C03633=1071.064,-119.142,443.657,172.455,21.905,153.991
C03634=1071.070,-118.892,443.648,172.457,21.906,153.991
C03635=1071.076,-118.643,443.638,172.457,21.907,153.991
C03636=1071.082,-118.393,443.629,172.459,21.908,153.991
C03637=1071.088,-118.143,443.619,172.461,21.909,153.991
C03638=1071.094,-117.893,443.610,172.463,21.910,153.991
C03639=1071.100,-117.643,443.601,172.464,21.911,153.990
C03640=1071.106,-117.393,443.591,172.466,21.912,153.990
C03641=1071.112,-117.143,443.582,172.468,21.913,153.990
C03642=1071.119,-116.893,443.572,172.469,21.914,153.990
C03643=1071.125,-116.644,443.563,172.471,21.915,153.990
C03644=1071.130,-116.395,443.553,172.473,21.916,153.990
C03645=1071.137,-116.145,443.544,172.475,21.917,153.990
C03646=1071.143,-115.895,443.535,172.476,21.918,153.990
C03647=1071.150,-115.646,443.525,172.478,21.919,153.990
C03648=1071.156,-115.396,443.516,172.479,21.920,153.990
C03649=1071.162,-115.146,443.506,172.480,21.921,153.990
C03650=1071.168,-114.896,443.497,172.482,21.922,153.990
C03651=1071.174,-114.646,443.487,172.484,21.923,153.990
C03652=1071.181,-114.367,443.476,172.486,21.924,153.990
C03653=1071.188,-114.087,443.466,172.488,21.925,153.989
C03654=1071.195,-113.808,443.455,172.490,21.927,153.989
C03655=1071.201,-113.528,443.443,172.492,21.927,153.989
C03656=1071.208,-113.278,443.434,172.493,21.929,153.989
C03657=1071.214,-113.029,443.424,172.495,21.930,153.989
C03658=1071.220,-112.779,443.415,172.497,21.931,153.989
C03659=1071.226,-112.529,443.405,172.498,21.932,153.989
C03660=1071.232,-112.280,443.396,172.500,21.933,153.989
C03661=1071.238,-112.030,443.386,172.502,21.934,153.989
C03662=1071.244,-111.780,443.377,172.502,21.935,153.989
C03663=1071.250,-111.531,443.367,172.504,21.936,153.989
C03664=1071.257,-111.281,443.357,172.506,21.937,153.989
C03665=1071.263,-111.032,443.347,172.508,21.938,153.989
C03666=1071.269,-110.782,443.338,172.509,21.939,153.989
C03667=1071.274,-110.532,443.328,172.511,21.940,153.989
C03668=1071.281,-110.282,443.318,172.512,21.942,153.989
C03669=1071.287,-110.032,443.309,172.514,21.942,153.989
C03670=1071.293,-109.782,443.299,172.516,21.944,153.989
C03671=1071.299,-109.533,443.289,172.517,21.945,153.989
C03672=1071.306,-109.283,443.279,172.519,21.946,153.989
C03673=1071.312,-109.034,443.270,172.521,21.947,153.989
C03674=1071.318,-108.784,443.260,172.523,21.948,153.989
C03675=1071.324,-108.534,443.250,172.524,21.950,153.989
C03676=1071.330,-108.284,443.241,172.526,21.950,153.988
C03677=1071.336,-108.035,443.230,172.527,21.952,153.988
C03678=1071.342,-107.785,443.220,172.529,21.953,153.988
C03679=1071.348,-107.535,443.211,172.531,21.954,153.988
C03680=1071.354,-107.285,443.201,172.532,21.955,153.988
C03681=1071.361,-107.035,443.192,172.533,21.956,153.988
C03682=1071.367,-106.786,443.181,172.535,21.957,153.988
C03683=1071.373,-106.536,443.171,172.536,21.959,153.988
C03684=1071.379,-106.286,443.162,172.538,21.960,153.988
C03685=1071.385,-106.037,443.152,172.540,21.961,153.988
C03686=1071.391,-105.787,443.142,172.541,21.962,153.988
C03687=1071.397,-105.537,443.132,172.543,21.964,153.988
C03688=1071.403,-105.287,443.122,172.545,21.964,153.988
C03689=1071.409,-105.038,443.113,172.546,21.966,153.988
C03690=1071.416,-104.788,443.102,172.548,21.967,153.988
C03691=1071.422,-104.538,443.092,172.550,21.968,153.988
C03692=1071.428,-104.288,443.082,172.551,21.969,153.988
C03693=1071.434,-104.039,443.072,172.553,21.971,153.988
C03694=1071.441,-103.789,443.062,172.554,21.972,153.988
C03695=1071.446,-103.539,443.052,172.556,21.973,153.988
C03696=1071.452,-103.290,443.042,172.558,21.974,153.988
C03697=1071.459,-103.040,443.032,172.559,21.976,153.988
C03698=1071.464,-102.790,443.022,172.561,21.977,153.988
C03699=1071.470,-102.541,443.012,172.563,21.978,153.988
C03700=1071.477,-102.291,443.002,172.564,21.979,153.988
C03701=1071.483,-102.041,442.993,172.566,21.981,153.988
C03702=1071.489,-101.791,442.982,172.568,21.982,153.988
C03703=1071.495,-101.542,442.972,172.569,21.983,153.988
C03704=1071.501,-101.292,442.963,172.571,21.985,153.988
C03705=1071.507,-101.042,442.952,172.573,21.986,153.988
C03706=1071.513,-100.792,442.942,172.574,21.987,153.988
C03707=1071.520,-100.543,442.932,172.576,21.988,153.988
C03708=1071.525,-100.293,442.921,172.577,21.990,153.988
C03709=1071.532,-100.043,442.912,172.579,21.991,153.988
C03710=1071.538,-99.794,442.902,172.580,21.992,153.988
C03711=1071.543,-99.543,442.891,172.581,21.993,153.988
C03712=1071.550,-99.294,442.881,172.583,21.994,153.988
C03713=1071.556,-99.045,442.872,172.584,21.996,153.988
C03714=1071.562,-98.795,442.861,172.586,21.997,153.988
C03715=1071.569,-98.545,442.851,172.588,21.998,153.988
C03716=1071.575,-98.263,442.839,172.590,22.000,153.988
C03717=1071.583,-97.981,442.828,172.592,22.001,153.988
C03718=1071.589,-97.699,442.817,172.593,22.003,153.988
C03719=1071.596,-97.417,442.805,172.595,22.004,153.988
C03720=1071.602,-97.167,442.795,172.596,22.006,153.988
C03721=1071.608,-96.918,442.784,172.598,22.007,153.988
C03722=1071.614,-96.668,442.775,172.600,22.008,153.988
C03723=1071.620,-96.418,442.764,172.601,22.010,153.988
C03724=1071.626,-96.169,442.754,172.603,22.011,153.988
C03725=1071.632,-95.919,442.743,172.604,22.012,153.988
C03726=1071.638,-95.670,442.732,172.606,22.014,153.988
C03727=1071.644,-95.420,442.723,172.608,22.015,153.988
C03728=1071.650,-95.170,442.712,172.609,22.017,153.988
C03729=1071.656,-94.920,442.702,172.611,22.018,153.988
C03730=1071.662,-94.670,442.691,172.612,22.019,153.988
C03731=1071.668,-94.421,442.682,172.614,22.021,153.988
C03732=1071.674,-94.171,442.671,172.615,22.022,153.988
C03733=1071.680,-93.921,442.661,172.617,22.023,153.988
C03734=1071.686,-93.672,442.650,172.619,22.025,153.988
C03735=1071.692,-93.423,442.640,172.620,22.027,153.988
C03736=1071.698,-93.172,442.629,172.622,22.028,153.988
C03737=1071.704,-92.922,442.619,172.623,22.030,153.988
C03738=1071.711,-92.673,442.608,172.625,22.031,153.988
C03739=1071.716,-92.423,442.598,172.626,22.032,153.988
C03740=1071.723,-92.174,442.588,172.628,22.034,153.988
C03741=1071.728,-91.924,442.578,172.630,22.035,153.988
C03742=1071.735,-91.674,442.567,172.631,22.036,153.989
C03743=1071.741,-91.424,442.556,172.633,22.038,153.989
C03744=1071.746,-91.174,442.546,172.634,22.039,153.989
C03745=1071.753,-90.925,442.536,172.636,22.041,153.989
C03746=1071.759,-90.676,442.525,172.637,22.042,153.989
C03747=1071.765,-90.426,442.515,172.639,22.044,153.989
C03748=1071.771,-90.176,442.504,172.640,22.045,153.989
C03749=1071.777,-89.926,442.493,172.642,22.047,153.989
C03750=1071.783,-89.676,442.484,172.644,22.048,153.989
C03751=1071.789,-89.427,442.473,172.645,22.049,153.989
C03752=1071.796,-89.177,442.462,172.647,22.051,153.989
C03753=1071.801,-88.927,442.451,172.648,22.053,153.989
C03754=1071.807,-88.677,442.441,172.650,22.054,153.989
C03755=1071.813,-88.428,442.431,172.651,22.055,153.989
C03756=1071.820,-88.178,442.420,172.653,22.057,153.989
C03757=1071.825,-87.928,442.409,172.654,22.059,153.989
C03758=1071.832,-87.679,442.399,172.656,22.060,153.989
C03759=1071.837,-87.429,442.388,172.658,22.061,153.989
C03760=1071.844,-87.179,442.378,172.659,22.063,153.989
C03761=1071.850,-86.930,442.367,172.661,22.064,153.989
C03762=1071.856,-86.680,442.357,172.662,22.066,153.989
C03763=1071.862,-86.431,442.346,172.664,22.068,153.989
C03764=1071.868,-86.180,442.335,172.665,22.069,153.989
C03765=1071.874,-85.931,442.324,172.667,22.070,153.989
C03766=1071.881,-85.682,442.314,172.668,22.072,153.989
C03767=1071.886,-85.432,442.303,172.670,22.074,153.990
C03768=1071.892,-85.181,442.292,172.671,22.075,153.990
C03769=1071.899,-84.932,442.282,172.673,22.076,153.990
C03770=1071.905,-84.683,442.271,172.675,22.078,153.990
C03771=1071.911,-84.433,442.260,172.676,22.080,153.990
C03772=1071.917,-84.183,442.250,172.678,22.081,153.990
C03773=1071.923,-83.934,442.239,172.679,22.082,153.990
C03774=1071.929,-83.683,442.228,172.681,22.084,153.990
C03775=1071.936,-83.434,442.218,172.682,22.086,153.990
C03776=1071.941,-83.184,442.207,172.684,22.087,153.990
C03777=1071.948,-82.934,442.196,172.685,22.088,153.990
C03778=1071.954,-82.685,442.186,172.687,22.090,153.990
C03779=1071.960,-82.436,442.175,172.689,22.092,153.990
C03780=1071.967,-82.156,442.163,172.691,22.093,153.990
C03781=1071.974,-81.877,442.150,172.692,22.095,153.990
C03782=1071.981,-81.597,442.138,172.694,22.097,153.990
C03783=1071.988,-81.317,442.127,172.696,22.099,153.990
C03784=1071.994,-81.067,442.116,172.698,22.100,153.990
C03785=1072.000,-80.818,442.105,172.699,22.102,153.990
C03786=1072.007,-80.568,442.094,172.701,22.104,153.991
C03787=1072.013,-80.318,442.083,172.702,22.105,153.991
C03788=1072.018,-80.069,442.073,172.704,22.107,153.991
C03789=1072.025,-79.819,442.061,172.705,22.108,153.991
C03790=1072.031,-79.569,442.051,172.707,22.110,153.991
C03791=1072.037,-79.320,442.040,172.708,22.112,153.991
C03792=1072.043,-79.070,442.029,172.710,22.113,153.991
C03793=1072.049,-78.820,442.018,172.711,22.115,153.991
C03794=1072.055,-78.571,442.007,172.713,22.116,153.991
C03795=1072.061,-78.321,441.996,172.714,22.118,153.991
C03796=1072.067,-78.071,441.985,172.716,22.120,153.991
C03797=1072.073,-77.821,441.974,172.717,22.121,153.991
C03798=1072.079,-77.571,441.963,172.719,22.123,153.992
C03799=1072.085,-77.322,441.952,172.720,22.124,153.992
C03800=1072.092,-77.072,441.941,172.722,22.126,153.992
C03801=1072.097,-76.822,441.930,172.723,22.128,153.992
C03802=1072.103,-76.573,441.920,172.725,22.130,153.992
C03803=1072.110,-76.323,441.908,172.726,22.131,153.992
C03804=1072.116,-76.074,441.897,172.728,22.133,153.992
C03805=1072.121,-75.824,441.886,172.729,22.134,153.992
C03806=1072.128,-75.574,441.875,172.731,22.136,153.992
C03807=1072.133,-75.325,441.864,172.732,22.138,153.992
C03808=1072.140,-75.075,441.853,172.734,22.140,153.992
C03809=1072.145,-74.825,441.842,172.735,22.141,153.992
C03810=1072.152,-74.575,441.830,172.737,22.143,153.993
C03811=1072.158,-74.325,441.820,172.738,22.144,153.993
C03812=1072.164,-74.076,441.809,172.741,22.147,153.993
C03813=1072.170,-73.826,441.797,172.742,22.148,153.993
C03814=1072.176,-73.577,441.786,172.743,22.150,153.993
C03815=1072.181,-73.327,441.775,172.745,22.152,153.993
C03816=1072.188,-73.077,441.764,172.746,22.154,153.993
C03817=1072.193,-72.828,441.753,172.748,22.155,153.993
C03818=1072.200,-72.577,441.742,172.749,22.157,153.993
C03819=1072.206,-72.329,441.730,172.751,22.159,153.993
C03820=1072.212,-72.079,441.719,172.752,22.160,153.993
C03821=1072.217,-71.829,441.707,172.754,22.162,153.994
C03822=1072.223,-71.579,441.696,172.755,22.164,153.994
C03823=1072.229,-71.330,441.685,172.757,22.165,153.994
C03824=1072.235,-71.080,441.674,172.758,22.167,153.994
C03825=1072.241,-70.831,441.663,172.759,22.169,153.994
C03826=1072.247,-70.580,441.651,172.761,22.171,153.994
C03827=1072.253,-70.331,441.639,172.762,22.173,153.994
C03828=1072.258,-70.082,441.628,172.764,22.175,153.994
C03829=1072.265,-69.832,441.617,172.765,22.176,153.995
C03830=1072.271,-69.582,441.606,172.767,22.178,153.995
C03831=1072.277,-69.332,441.594,172.768,22.180,153.995
C03832=1072.283,-69.083,441.583,172.770,22.182,153.995
C03833=1072.289,-68.832,441.572,172.772,22.184,153.995
C03834=1072.294,-68.583,441.561,172.774,22.185,153.995
C03835=1072.300,-68.334,441.549,172.775,22.187,153.995
C03836=1072.307,-68.084,441.538,172.776,22.189,153.995
C03837=1072.312,-67.834,441.527,172.778,22.191,153.995
C03838=1072.319,-67.585,441.515,172.779,22.193,153.995
C03839=1072.324,-67.335,441.504,172.781,22.194,153.996
C03840=1072.330,-67.085,441.492,172.782,22.196,153.996
C03841=1072.336,-66.836,441.481,172.784,22.198,153.996
C03842=1072.343,-66.586,441.469,172.785,22.200,153.996
C03843=1072.349,-66.337,441.458,172.786,22.202,153.996
C03844=1072.355,-66.059,441.445,172.788,22.204,153.996
C03845=1072.362,-65.782,441.432,172.790,22.206,153.996
C03846=1072.369,-65.504,441.419,172.792,22.208,153.996
C03847=1072.376,-65.227,441.407,172.793,22.210,153.997
C03848=1072.381,-64.977,441.395,172.794,22.212,153.997
C03849=1072.387,-64.727,441.384,172.796,22.214,153.997
C03850=1072.393,-64.478,441.373,172.797,22.215,153.997
C03851=1072.400,-64.228,441.361,172.799,22.217,153.997
C03852=1072.405,-63.978,441.349,172.801,22.219,153.997
C03853=1072.411,-63.728,441.338,172.802,22.221,153.997
C03854=1072.417,-63.479,441.326,172.804,22.223,153.997
C03855=1072.423,-63.229,441.315,172.805,22.225,153.998
C03856=1072.429,-62.980,441.304,172.807,22.227,153.998
C03857=1072.435,-62.730,441.292,172.808,22.229,153.998
C03858=1072.441,-62.481,441.280,172.810,22.230,153.998
C03859=1072.447,-62.231,441.269,172.811,22.232,153.998
C03860=1072.454,-61.981,441.257,172.812,22.234,153.998
C03861=1072.459,-61.731,441.245,172.814,22.236,153.998
C03862=1072.466,-61.482,441.233,172.815,22.238,153.999
C03863=1072.472,-61.232,441.223,172.817,22.240,153.999
C03864=1072.478,-60.983,441.211,172.818,22.242,153.999
C03865=1072.483,-60.733,441.199,172.820,22.243,153.999
C03866=1072.490,-60.483,441.187,172.821,22.245,153.999
C03867=1072.496,-60.233,441.176,172.823,22.247,153.999
C03868=1072.501,-59.984,441.164,172.825,22.249,153.999
C03869=1072.508,-59.734,441.152,172.826,22.251,153.999
C03870=1072.514,-59.485,441.141,172.828,22.253,154.000
C03871=1072.520,-59.235,441.129,172.829,22.255,154.000
C03872=1072.526,-58.985,441.117,172.830,22.257,154.000
C03873=1072.532,-58.736,441.106,172.832,22.258,154.000
C03874=1072.538,-58.486,441.094,172.833,22.260,154.000
C03875=1072.544,-58.236,441.082,172.835,22.262,154.000
C03876=1072.550,-57.987,441.070,172.836,22.264,154.000
C03877=1072.557,-57.737,441.059,172.838,22.266,154.001
C03878=1072.563,-57.488,441.047,172.839,22.268,154.001
C03879=1072.569,-57.238,441.035,172.840,22.270,154.001
C03880=1072.575,-56.988,441.024,172.842,22.272,154.001
C03881=1072.581,-56.739,441.012,172.844,22.274,154.001
C03882=1072.587,-56.489,441.000,172.846,22.276,154.001
C03883=1072.593,-56.239,440.988,172.847,22.278,154.001
C03884=1072.599,-55.990,440.977,172.848,22.280,154.002
C03885=1072.605,-55.740,440.965,172.850,22.281,154.002
C03886=1072.612,-55.490,440.953,172.851,22.283,154.002
C03887=1072.618,-55.241,440.941,172.853,22.285,154.002
C03888=1072.624,-54.991,440.929,172.854,22.287,154.002
C03889=1072.630,-54.741,440.917,172.856,22.289,154.002
C03890=1072.637,-54.491,440.905,172.857,22.291,154.002
C03891=1072.642,-54.242,440.893,172.858,22.293,154.002
C03892=1072.648,-53.992,440.882,172.860,22.295,154.003
C03893=1072.655,-53.743,440.870,172.861,22.296,154.003
C03894=1072.660,-53.493,440.858,172.863,22.298,154.003
C03895=1072.667,-53.244,440.846,172.865,22.301,154.003
C03896=1072.673,-52.994,440.835,172.866,22.303,154.003
C03897=1072.679,-52.744,440.822,172.868,22.304,154.003
C03898=1072.685,-52.495,440.810,172.869,22.306,154.003
C03899=1072.691,-52.245,440.798,172.870,22.308,154.004
C03900=1072.697,-51.995,440.787,172.872,22.310,154.004
C03901=1072.703,-51.746,440.775,172.873,22.312,154.004
C03902=1072.709,-51.496,440.763,172.875,22.314,154.004
C03903=1072.716,-51.246,440.751,172.876,22.316,154.004
C03904=1072.723,-50.997,440.739,172.878,22.318,154.004
C03905=1072.728,-50.746,440.727,172.879,22.320,154.005
C03906=1072.734,-50.497,440.715,172.880,22.322,154.005
C03907=1072.740,-50.248,440.703,172.883,22.324,154.005
C03908=1072.747,-49.972,440.690,172.884,22.326,154.005
C03909=1072.754,-49.696,440.676,172.885,22.328,154.005
C03910=1072.760,-49.419,440.662,172.887,22.330,154.005
C03911=1072.766,-49.144,440.649,172.889,22.333,154.006
C03912=1072.773,-48.894,440.638,172.890,22.335,154.006
C03913=1072.779,-48.644,440.625,172.892,22.337,154.006
C03914=1072.785,-48.394,440.613,172.893,22.339,154.006
C03915=1072.791,-48.145,440.601,172.894,22.341,154.006
C03916=1072.797,-47.895,440.588,172.896,22.343,154.007
C03917=1072.802,-47.645,440.576,172.897,22.345,154.007
C03918=1072.809,-47.396,440.564,172.898,22.347,154.007
C03919=1072.814,-47.147,440.552,172.900,22.349,154.007
C03920=1072.820,-46.897,440.539,172.902,22.351,154.007
C03921=1072.827,-46.647,440.527,172.903,22.354,154.007
C03922=1072.832,-46.398,440.515,172.905,22.356,154.008
C03923=1072.838,-46.148,440.502,172.906,22.358,154.008
C03924=1072.845,-45.898,440.490,172.908,22.360,154.008
C03925=1072.851,-45.649,440.478,172.909,22.362,154.008
C03926=1072.856,-45.399,440.466,172.910,22.364,154.008
C03927=1072.862,-45.149,440.454,172.912,22.366,154.008
C03928=1072.868,-44.899,440.442,172.913,22.368,154.009
C03929=1072.874,-44.649,440.429,172.914,22.370,154.009
C03930=1072.880,-44.401,440.418,172.916,22.372,154.009
C03931=1072.886,-44.151,440.405,172.918,22.375,154.009
C03932=1072.892,-43.901,440.392,172.919,22.376,154.009
C03933=1072.898,-43.652,440.379,172.921,22.378,154.009
C03934=1072.905,-43.402,440.367,172.922,22.381,154.010
C03935=1072.910,-43.153,440.355,172.923,22.383,154.010
C03936=1072.916,-42.903,440.343,172.925,22.385,154.010
C03937=1072.923,-42.653,440.331,172.926,22.387,154.010
C03938=1072.929,-42.403,440.318,172.927,22.389,154.010
C03939=1072.935,-42.154,440.306,172.929,22.391,154.011
C03940=1072.941,-41.905,440.294,172.930,22.393,154.011
C03941=1072.947,-41.655,440.281,172.932,22.395,154.011
C03942=1072.952,-41.405,440.269,172.934,22.398,154.011
C03943=1072.958,-41.155,440.256,172.935,22.400,154.011
C03944=1072.965,-40.905,440.244,172.937,22.401,154.011
C03945=1072.971,-40.656,440.232,172.938,22.403,154.012
C03946=1072.977,-40.406,440.219,172.939,22.406,154.012
C03947=1072.982,-40.157,440.206,172.941,22.408,154.012
C03948=1072.989,-39.908,440.194,172.942,22.410,154.012
C03949=1072.995,-39.658,440.182,172.943,22.412,154.012
C03950=1073.001,-39.408,440.169,172.945,22.414,154.013
C03951=1073.007,-39.158,440.157,172.946,22.416,154.013
C03952=1073.014,-38.909,440.144,172.948,22.418,154.013
C03953=1073.020,-38.659,440.132,172.950,22.421,154.013
C03954=1073.025,-38.410,440.119,172.951,22.423,154.013
C03955=1073.031,-38.160,440.107,172.952,22.425,154.014
C03956=1073.037,-37.910,440.094,172.954,22.427,154.014
C03957=1073.043,-37.660,440.082,172.955,22.429,154.014
C03958=1073.049,-37.411,440.068,172.956,22.431,154.014
C03959=1073.055,-37.161,440.056,172.958,22.433,154.014
C03960=1073.060,-36.912,440.044,172.959,22.436,154.015
C03961=1073.067,-36.662,440.032,172.960,22.438,154.015
C03962=1073.073,-36.413,440.018,172.963,22.440,154.015
C03963=1073.079,-36.163,440.006,172.964,22.442,154.015
C03964=1073.085,-35.913,439.993,172.965,22.444,154.015
C03965=1073.091,-35.663,439.981,172.967,22.447,154.016
C03966=1073.097,-35.414,439.968,172.968,22.449,154.016
C03967=1073.102,-35.165,439.955,172.969,22.451,154.016
C03968=1073.108,-34.915,439.943,172.971,22.453,154.016
C03969=1073.114,-34.666,439.930,172.972,22.455,154.016
C03970=1073.120,-34.416,439.917,172.973,22.457,154.017
C03971=1073.126,-34.166,439.904,172.975,22.459,154.017
C03972=1073.132,-33.890,439.890,172.977,22.462,154.017
C03973=1073.140,-33.614,439.876,172.978,22.465,154.017
C03974=1073.146,-33.339,439.862,172.979,22.467,154.017
C03975=1073.152,-33.063,439.849,172.982,22.469,154.018
C03976=1073.159,-32.814,439.835,172.983,22.471,154.018
C03977=1073.165,-32.564,439.823,172.984,22.474,154.018
C03978=1073.171,-32.315,439.810,172.986,22.476,154.018
C03979=1073.177,-32.065,439.797,172.987,22.478,154.019
C03980=1073.183,-31.815,439.784,172.988,22.480,154.019
C03981=1073.189,-31.566,439.771,172.990,22.483,154.019
C03982=1073.195,-31.316,439.759,172.991,22.484,154.019
C03983=1073.201,-31.066,439.746,172.993,22.487,154.019
C03984=1073.207,-30.817,439.733,172.994,22.489,154.020
C03985=1073.213,-30.567,439.720,172.996,22.492,154.020
C03986=1073.219,-30.318,439.707,172.997,22.494,154.020
C03987=1073.225,-30.068,439.694,172.998,22.496,154.020
C03988=1073.231,-29.819,439.681,173.000,22.498,154.020
C03989=1073.237,-29.569,439.669,173.001,22.500,154.021
C03990=1073.243,-29.319,439.655,173.002,22.502,154.021
C03991=1073.249,-29.070,439.643,173.004,22.504,154.021
C03992=1073.255,-28.820,439.630,173.006,22.507,154.021
C03993=1073.261,-28.570,439.617,173.007,22.509,154.021
C03994=1073.267,-28.321,439.604,173.009,22.511,154.022
C03995=1073.273,-28.071,439.591,173.010,22.513,154.022
C03996=1073.279,-27.821,439.579,173.011,22.516,154.022
C03997=1073.285,-27.572,439.565,173.013,22.518,154.022
C03998=1073.291,-27.322,439.553,173.014,22.520,154.023
C03999=1073.298,-27.073,439.539,173.015,22.522,154.023
C04000=1073.303,-26.823,439.526,173.017,22.525,154.023
C04001=1073.309,-26.574,439.513,173.019,22.527,154.023
C04002=1073.315,-26.324,439.500,173.020,22.529,154.023
C04003=1073.321,-26.074,439.487,173.021,22.532,154.024
C04004=1073.327,-25.825,439.474,173.023,22.534,154.024
C04005=1073.332,-25.575,439.461,173.024,22.536,154.024
C04006=1073.339,-25.326,439.448,173.025,22.539,154.024
C04007=1073.345,-25.076,439.435,173.027,22.540,154.025
C04008=1073.351,-24.827,439.422,173.028,22.543,154.025
C04009=1073.356,-24.577,439.408,173.029,22.545,154.025
C04010=1073.362,-24.327,439.395,173.031,22.548,154.025
C04011=1073.368,-24.078,439.382,173.033,22.550,154.026
C04012=1073.374,-23.828,439.369,173.034,22.552,154.026
C04013=1073.380,-23.578,439.356,173.035,22.554,154.026
C04014=1073.386,-23.329,439.342,173.037,22.557,154.026
C04015=1073.392,-23.079,439.330,173.038,22.559,154.026
C04016=1073.398,-22.830,439.317,173.039,22.561,154.027
C04017=1073.404,-22.580,439.303,173.041,22.563,154.027
C04018=1073.409,-22.330,439.290,173.042,22.566,154.027
C04019=1073.416,-22.081,439.277,173.044,22.568,154.027
C04020=1073.422,-21.832,439.264,173.045,22.570,154.028
C04021=1073.427,-21.582,439.250,173.047,22.573,154.028
C04022=1073.433,-21.332,439.237,173.048,22.575,154.028
C04023=1073.440,-21.083,439.224,173.049,22.577,154.028
C04024=1073.445,-20.833,439.211,173.051,22.580,154.029
C04025=1073.451,-20.584,439.197,173.052,22.582,154.029
C04026=1073.457,-20.334,439.184,173.053,22.584,154.029
C04027=1073.464,-20.085,439.171,173.055,22.587,154.029
C04028=1073.469,-19.834,439.157,173.057,22.589,154.029
C04029=1073.475,-19.585,439.144,173.058,22.591,154.030
C04030=1073.482,-19.336,439.131,173.059,22.594,154.030
C04031=1073.488,-19.087,439.118,173.061,22.596,154.030
C04032=1073.493,-18.836,439.104,173.062,22.598,154.030
C04033=1073.499,-18.587,439.091,173.063,22.600,154.031
C04034=1073.505,-18.338,439.078,173.065,22.602,154.031
C04035=1073.511,-18.088,439.064,173.066,22.605,154.031
C04036=1073.518,-17.811,439.049,173.068,22.608,154.031
C04037=1073.525,-17.535,439.035,173.069,22.610,154.032
C04038=1073.531,-17.258,439.020,173.070,22.613,154.032
C04039=1073.538,-16.982,439.006,173.073,22.615,154.032
C04040=1073.543,-16.732,438.992,173.074,22.618,154.032
C04041=1073.550,-16.482,438.978,173.075,22.620,154.033
C04042=1073.556,-16.233,438.965,173.076,22.622,154.033
C04043=1073.562,-15.984,438.951,173.078,22.625,154.033
C04044=1073.568,-15.734,438.938,173.079,22.627,154.033
C04045=1073.574,-15.484,438.925,173.081,22.629,154.034
C04046=1073.579,-15.235,438.911,173.082,22.632,154.034
C04047=1073.586,-14.985,438.898,173.084,22.634,154.034
C04048=1073.592,-14.735,438.884,173.085,22.636,154.034
C04049=1073.598,-14.486,438.871,173.086,22.639,154.035
C04050=1073.603,-14.237,438.857,173.088,22.641,154.035
C04051=1073.610,-13.987,438.843,173.089,22.643,154.035
C04052=1073.615,-13.738,438.830,173.090,22.645,154.035
C04053=1073.621,-13.488,438.816,173.092,22.648,154.036
C04054=1073.627,-13.239,438.802,173.094,22.651,154.036
C04055=1073.633,-12.988,438.790,173.095,22.653,154.036
C04056=1073.639,-12.739,438.776,173.096,22.655,154.036
C04057=1073.645,-12.489,438.762,173.098,22.658,154.037
C04058=1073.651,-12.240,438.749,173.099,22.660,154.037
C04059=1073.657,-11.991,438.735,173.100,22.662,154.037
C04060=1073.662,-11.741,438.721,173.101,22.664,154.037
C04061=1073.668,-11.491,438.707,173.103,22.667,154.038
C04062=1073.675,-11.241,438.694,173.105,22.670,154.038
C04063=1073.680,-10.992,438.680,173.106,22.672,154.038
C04064=1073.686,-10.743,438.667,173.107,22.675,154.038
C04065=1073.692,-10.493,438.653,173.109,22.676,154.038
C04066=1073.698,-10.243,438.639,173.110,22.679,154.039
C04067=1073.704,-9.994,438.625,173.111,22.681,154.039
C04068=1073.710,-9.744,438.612,173.112,22.684,154.039
C04069=1073.716,-9.495,438.598,173.114,22.686,154.040
C04070=1073.721,-9.246,438.584,173.116,22.688,154.040
C04071=1073.728,-8.996,438.570,173.117,22.691,154.040
C04072=1073.734,-8.746,438.556,173.119,22.693,154.040
C04073=1073.740,-8.497,438.543,173.120,22.696,154.041
C04074=1073.745,-8.247,438.529,173.121,22.698,154.041
C04075=1073.752,-7.997,438.515,173.122,22.700,154.041
C04076=1073.758,-7.748,438.502,173.124,22.703,154.041
C04077=1073.763,-7.498,438.488,173.125,22.705,154.042
C04078=1073.769,-7.249,438.474,173.127,22.708,154.042
C04079=1073.775,-6.999,438.460,173.128,22.710,154.042
C04080=1073.782,-6.750,438.446,173.130,22.712,154.042
C04081=1073.787,-6.500,438.432,173.131,22.715,154.043
C04082=1073.793,-6.251,438.418,173.132,22.717,154.043
C04083=1073.800,-6.001,438.405,173.134,22.720,154.043
C04084=1073.805,-5.751,438.391,173.135,22.722,154.043
C04085=1073.811,-5.502,438.378,173.137,22.724,154.044
C04086=1073.817,-5.253,438.363,173.138,22.727,154.044
C04087=1073.823,-5.003,438.349,173.140,22.729,154.044
C04088=1073.830,-4.754,438.336,173.141,22.732,154.044
C04089=1073.835,-4.504,438.322,173.142,22.734,154.045
C04090=1073.841,-4.254,438.308,173.143,22.737,154.045
C04091=1073.848,-4.005,438.294,173.145,22.738,154.045
C04092=1073.853,-3.756,438.280,173.146,22.741,154.045
C04093=1073.860,-3.506,438.266,173.148,22.744,154.046
C04094=1073.865,-3.256,438.252,173.149,22.746,154.046
C04095=1073.871,-3.007,438.238,173.151,22.749,154.046
C04096=1073.877,-2.757,438.224,173.152,22.751,154.047
C04097=1073.883,-2.507,438.209,173.153,22.753,154.047
C04098=1073.888,-2.258,438.196,173.154,22.756,154.047
C04099=1073.895,-2.009,438.182,173.156,22.758,154.047
C04100=1073.901,-1.730,438.166,173.158,22.761,154.048
C04101=1073.907,-1.453,438.150,173.159,22.764,154.048
C04102=1073.914,-1.174,438.134,173.160,22.766,154.048
C04103=1073.920,-0.895,438.119,173.162,22.769,154.049
C04104=1073.926,-0.646,438.104,173.163,22.772,154.049
C04105=1073.932,-0.397,438.090,173.165,22.774,154.049
C04106=1073.938,-0.147,438.076,173.166,22.777,154.049
C04107=1073.944,0.102,438.062,173.167,22.779,154.050
C04108=1073.950,0.352,438.048,173.168,22.782,154.050
C04109=1073.956,0.602,438.034,173.171,22.784,154.050
C04110=1073.962,0.851,438.020,173.172,22.786,154.050
C04111=1073.967,1.100,438.006,173.173,22.789,154.051
C04112=1073.973,1.349,437.991,173.175,22.791,154.051
C04113=1073.979,1.600,437.977,173.176,22.794,154.051
C04114=1073.984,1.849,437.963,173.177,22.796,154.052
C04115=1073.990,2.098,437.948,173.178,22.799,154.052
C04116=1073.996,2.349,437.934,173.180,22.801,154.052
C04117=1074.002,2.597,437.920,173.182,22.804,154.052
C04118=1074.008,2.847,437.906,173.183,22.806,154.053
C04119=1074.015,3.096,437.891,173.184,22.809,154.053
C04120=1074.020,3.346,437.878,173.185,22.811,154.053
C04121=1074.026,3.596,437.863,173.187,22.814,154.054
C04122=1074.032,3.845,437.849,173.188,22.816,154.054
C04123=1074.037,4.095,437.835,173.189,22.818,154.054
C04124=1074.044,4.344,437.820,173.191,22.821,154.054
C04125=1074.049,4.594,437.806,173.193,22.824,154.055
C04126=1074.055,4.843,437.791,173.194,22.826,154.055
C04127=1074.061,5.093,437.777,173.195,22.829,154.055
C04128=1074.067,5.342,437.763,173.196,22.831,154.055
C04129=1074.073,5.592,437.748,173.198,22.833,154.056
C04130=1074.079,5.841,437.734,173.199,22.836,154.056
C04131=1074.084,6.091,437.720,173.201,22.839,154.056
C04132=1074.091,6.341,437.705,173.202,22.841,154.057
C04133=1074.096,6.590,437.691,173.204,22.844,154.057
C04134=1074.102,6.840,437.676,173.205,22.846,154.057
C04135=1074.109,7.089,437.662,173.206,22.848,154.057
C04136=1074.115,7.339,437.648,173.208,22.850,154.058
C04137=1074.121,7.588,437.633,173.209,22.853,154.058
C04138=1074.126,7.837,437.620,173.211,22.856,154.058
C04139=1074.133,8.087,437.605,173.212,22.858,154.058
C04140=1074.138,8.337,437.591,173.213,22.860,154.059
C04141=1074.145,8.586,437.576,173.215,22.863,154.059
C04142=1074.150,8.835,437.561,173.216,22.865,154.059
C04143=1074.156,9.085,437.547,173.217,22.868,154.060
C04144=1074.162,9.334,437.532,173.218,22.870,154.060
C04145=1074.169,9.584,437.517,173.221,22.873,154.060
C04146=1074.174,9.834,437.504,173.222,22.875,154.060
C04147=1074.180,10.083,437.489,173.223,22.878,154.061
C04148=1074.186,10.332,437.474,173.224,22.880,154.061
C04149=1074.192,10.583,437.460,173.226,22.883,154.061
C04150=1074.198,10.831,437.445,173.227,22.885,154.062
C04151=1074.204,11.081,437.430,173.228,22.888,154.062
C04152=1074.210,11.331,437.416,173.229,22.890,154.062
C04153=1074.216,11.580,437.402,173.232,22.893,154.062
C04154=1074.222,11.829,437.387,173.233,22.895,154.063
C04155=1074.228,12.080,437.373,173.234,22.898,154.063
C04156=1074.234,12.329,437.358,173.235,22.900,154.063
C04157=1074.240,12.579,437.343,173.237,22.903,154.063
C04158=1074.245,12.827,437.328,173.238,22.905,154.064
C04159=1074.251,13.078,437.314,173.239,22.907,154.064
C04160=1074.257,13.327,437.299,173.241,22.910,154.064
C04161=1074.264,13.576,437.284,173.243,22.912,154.064
C04162=1074.269,13.825,437.270,173.244,22.915,154.065
C04163=1074.276,14.076,437.255,173.245,22.917,154.065
C04164=1074.282,14.355,437.239,173.246,22.920,154.065
C04165=1074.289,14.636,437.223,173.249,22.923,154.066
C04166=1074.296,14.915,437.205,173.250,22.925,154.066
C04167=1074.303,15.196,437.189,173.252,22.929,154.066
C04168=1074.308,15.445,437.174,173.253,22.931,154.067
C04169=1074.314,15.695,437.160,173.254,22.934,154.067
C04170=1074.320,15.944,437.145,173.256,22.936,154.067
C04171=1074.326,16.194,437.130,173.257,22.938,154.067
C04172=1074.332,16.443,437.116,173.258,22.941,154.068
C04173=1074.338,16.693,437.100,173.260,22.944,154.068
C04174=1074.343,16.942,437.085,173.261,22.946,154.068
C04175=1074.349,17.192,437.071,173.263,22.948,154.069
C04176=1074.355,17.441,437.057,173.264,22.951,154.069
C04177=1074.361,17.691,437.041,173.265,22.953,154.069
C04178=1074.367,17.940,437.026,173.267,22.956,154.069
C04179=1074.373,18.190,437.012,173.268,22.958,154.070
C04180=1074.379,18.439,436.997,173.270,22.961,154.070
C04181=1074.384,18.689,436.981,173.271,22.963,154.070
C04182=1074.391,18.938,436.966,173.272,22.966,154.071
C04183=1074.397,19.187,436.952,173.274,22.969,154.071
C04184=1074.402,19.437,436.936,173.275,22.971,154.071
C04185=1074.408,19.686,436.922,173.276,22.974,154.072
C04186=1074.414,19.936,436.907,173.277,22.976,154.072
C04187=1074.421,20.185,436.892,173.280,22.979,154.072
C04188=1074.425,20.435,436.877,173.281,22.981,154.072
C04189=1074.432,20.685,436.862,173.282,22.984,154.073
C04190=1074.438,20.934,436.848,173.283,22.986,154.073
C04191=1074.443,21.184,436.832,173.285,22.989,154.073
C04192=1074.450,21.434,436.817,173.286,22.991,154.074
C04193=1074.455,21.683,436.802,173.288,22.994,154.074
C04194=1074.461,21.932,436.787,173.289,22.996,154.074
C04195=1074.467,22.181,436.772,173.291,22.999,154.074
C04196=1074.473,22.431,436.756,173.292,23.002,154.075
C04197=1074.479,22.680,436.741,173.293,23.004,154.075
C04198=1074.484,22.930,436.726,173.294,23.007,154.075
C04199=1074.491,23.179,436.711,173.295,23.009,154.076
C04200=1074.496,23.428,436.697,173.298,23.012,154.076
C04201=1074.502,23.678,436.681,173.299,23.014,154.076
C04202=1074.508,23.928,436.666,173.300,23.017,154.076
C04203=1074.514,24.177,436.651,173.301,23.019,154.077
C04204=1074.520,24.427,436.636,173.303,23.022,154.077
C04205=1074.526,24.677,436.621,173.304,23.024,154.077
C04206=1074.531,24.926,436.606,173.306,23.027,154.078
C04207=1074.538,25.175,436.591,173.307,23.029,154.078
C04208=1074.543,25.424,436.575,173.308,23.032,154.078
C04209=1074.549,25.674,436.560,173.310,23.035,154.079
C04210=1074.555,25.924,436.545,173.311,23.037,154.079
C04211=1074.561,26.173,436.530,173.312,23.039,154.079
C04212=1074.567,26.423,436.515,173.314,23.042,154.079
C04213=1074.573,26.672,436.500,173.316,23.045,154.080
C04214=1074.580,26.921,436.484,173.317,23.047,154.080
C04215=1074.585,27.171,436.469,173.318,23.050,154.080
C04216=1074.591,27.420,436.454,173.320,23.052,154.081
C04217=1074.597,27.670,436.438,173.321,23.054,154.081
C04218=1074.602,27.919,436.424,173.322,23.057,154.081
C04219=1074.608,28.169,436.408,173.324,23.060,154.081
C04220=1074.615,28.418,436.393,173.326,23.062,154.082
C04221=1074.620,28.667,436.377,173.327,23.065,154.082
C04222=1074.626,28.917,436.362,173.328,23.067,154.082
C04223=1074.632,29.167,436.347,173.329,23.070,154.083
C04224=1074.637,29.416,436.331,173.330,23.072,154.083
C04225=1074.644,29.665,436.316,173.333,23.075,154.083
C04226=1074.649,29.915,436.301,173.334,23.077,154.083
C04227=1074.655,30.164,436.285,173.335,23.080,154.084
C04228=1074.661,30.446,436.268,173.336,23.083,154.084
C04229=1074.668,30.728,436.251,173.338,23.086,154.084
C04230=1074.674,31.009,436.233,173.340,23.089,154.085
C04231=1074.681,31.290,436.215,173.342,23.092,154.085
C04232=1074.687,31.540,436.200,173.343,23.094,154.085
C04233=1074.694,31.789,436.184,173.344,23.097,154.086
C04234=1074.699,32.039,436.169,173.345,23.099,154.086
C04235=1074.704,32.289,436.154,173.347,23.102,154.086
C04236=1074.711,32.538,436.138,173.349,23.104,154.087
C04237=1074.717,32.788,436.122,173.350,23.107,154.087
C04238=1074.722,33.037,436.107,173.351,23.109,154.087
C04239=1074.728,33.286,436.092,173.352,23.112,154.088
C04240=1074.734,33.536,436.076,173.354,23.115,154.088
C04241=1074.740,33.786,436.060,173.355,23.117,154.088
C04242=1074.746,34.034,436.045,173.357,23.120,154.088
C04243=1074.751,34.284,436.030,173.358,23.122,154.089
C04244=1074.757,34.533,436.013,173.360,23.125,154.089
C04245=1074.764,34.783,435.998,173.361,23.127,154.089
C04246=1074.769,35.032,435.983,173.362,23.130,154.090
C04247=1074.775,35.282,435.967,173.363,23.133,154.090
C04248=1074.781,35.531,435.952,173.366,23.135,154.090
C04249=1074.787,35.781,435.936,173.367,23.138,154.091
C04250=1074.793,36.031,435.920,173.368,23.140,154.091
C04251=1074.799,36.279,435.905,173.369,23.143,154.091
C04252=1074.804,36.529,435.889,173.371,23.145,154.091
C04253=1074.810,36.778,435.873,173.372,23.147,154.092
C04254=1074.817,37.028,435.858,173.374,23.150,154.092
C04255=1074.823,37.277,435.842,173.375,23.153,154.092
C04256=1074.828,37.527,435.827,173.377,23.155,154.092
C04257=1074.834,37.776,435.810,173.378,23.158,154.093
C04258=1074.840,38.026,435.796,173.379,23.160,154.093
C04259=1074.846,38.275,435.779,173.380,23.163,154.093
C04260=1074.852,38.525,435.764,173.383,23.166,154.094
C04261=1074.857,38.774,435.748,173.384,23.168,154.094
C04262=1074.863,39.023,435.732,173.385,23.171,154.094
C04263=1074.869,39.273,435.716,173.386,23.173,154.095
C04264=1074.875,39.522,435.700,173.387,23.176,154.095
C04265=1074.881,39.772,435.685,173.390,23.179,154.095
C04266=1074.886,40.021,435.669,173.391,23.181,154.096
C04267=1074.892,40.270,435.653,173.392,23.184,154.096
C04268=1074.898,40.520,435.637,173.393,23.186,154.096
C04269=1074.904,40.769,435.621,173.395,23.189,154.097
C04270=1074.910,41.019,435.605,173.396,23.191,154.097
C04271=1074.915,41.268,435.589,173.398,23.194,154.097
C04272=1074.921,41.517,435.573,173.399,23.197,154.097
C04273=1074.927,41.767,435.558,173.401,23.199,154.098
C04274=1074.933,42.016,435.542,173.402,23.201,154.098
C04275=1074.939,42.266,435.526,173.403,23.204,154.098
C04276=1074.945,42.515,435.510,173.405,23.207,154.099
C04277=1074.951,42.765,435.494,173.406,23.210,154.099
C04278=1074.956,43.013,435.478,173.408,23.212,154.099
C04279=1074.962,43.263,435.463,173.409,23.214,154.099
C04280=1074.968,43.513,435.446,173.410,23.217,154.100
C04281=1074.974,43.762,435.430,173.412,23.219,154.100
C04282=1074.979,44.012,435.414,173.414,23.223,154.100
C04283=1074.985,44.261,435.398,173.415,23.225,154.101
C04284=1074.991,44.511,435.382,173.416,23.227,154.101
C04285=1074.997,44.759,435.366,173.417,23.230,154.101
C04286=1075.002,45.009,435.351,173.419,23.233,154.102
C04287=1075.008,45.259,435.334,173.421,23.235,154.102
C04288=1075.014,45.508,435.318,173.422,23.238,154.102
C04289=1075.020,45.757,435.302,173.423,23.240,154.103
C04290=1075.025,46.008,435.286,173.425,23.243,154.103
C04291=1075.030,46.256,435.270,173.426,23.246,154.103
C04292=1075.037,46.538,435.251,173.428,23.248,154.104
C04293=1075.043,46.819,435.233,173.429,23.251,154.104
C04294=1075.050,47.101,435.215,173.431,23.255,154.104
C04295=1075.056,47.382,435.196,173.432,23.257,154.105
C04296=1075.062,47.632,435.180,173.434,23.260,154.105
C04297=1075.068,47.882,435.164,173.436,23.263,154.105
C04298=1075.074,48.131,435.148,173.437,23.265,154.106
C04299=1075.080,48.380,435.132,173.438,23.268,154.106
C04300=1075.086,48.630,435.116,173.439,23.270,154.106
C04301=1075.092,48.879,435.099,173.441,23.273,154.106
C04302=1075.097,49.128,435.084,173.443,23.276,154.107
C04303=1075.102,49.377,435.067,173.444,23.278,154.107
C04304=1075.108,49.627,435.051,173.445,23.281,154.107
C04305=1075.114,49.877,435.035,173.447,23.283,154.108
C04306=1075.120,50.126,435.019,173.448,23.286,154.108
C04307=1075.126,50.375,435.002,173.450,23.289,154.108
C04308=1075.132,50.625,434.986,173.451,23.291,154.109
C04309=1075.137,50.874,434.969,173.453,23.294,154.109
C04310=1075.143,51.124,434.953,173.454,23.296,154.109
C04311=1075.149,51.373,434.937,173.455,23.299,154.109
C04312=1075.155,51.623,434.921,173.457,23.302,154.110
C04313=1075.161,51.872,434.904,173.458,23.304,154.110
C04314=1075.167,52.121,434.888,173.460,23.307,154.110
C04315=1075.172,52.371,434.871,173.461,23.309,154.111
C04316=1075.178,52.620,434.855,173.462,23.311,154.111
C04317=1075.184,52.870,434.839,173.464,23.314,154.111
C04318=1075.190,53.119,434.822,173.466,23.317,154.112
C04319=1075.196,53.368,434.806,173.467,23.320,154.112
C04320=1075.201,53.618,434.789,173.468,23.322,154.112
C04321=1075.207,53.867,434.773,173.469,23.324,154.113
C04322=1075.213,54.117,434.757,173.472,23.327,154.113
C04323=1075.219,54.366,434.741,173.473,23.330,154.113
C04324=1075.225,54.615,434.724,173.474,23.332,154.113
C04325=1075.230,54.865,434.707,173.475,23.335,154.114
C04326=1075.236,55.114,434.691,173.478,23.338,154.114
C04327=1075.242,55.364,434.675,173.479,23.340,154.114
C04328=1075.248,55.613,434.659,173.480,23.343,154.115
C04329=1075.253,55.862,434.641,173.481,23.345,154.115
C04330=1075.259,56.111,434.625,173.483,23.347,154.115
C04331=1075.265,56.361,434.609,173.485,23.350,154.115
C04332=1075.271,56.610,434.592,173.486,23.353,154.116
C04333=1075.276,56.860,434.575,173.487,23.356,154.116
C04334=1075.282,57.109,434.559,173.489,23.358,154.116
C04335=1075.288,57.358,434.543,173.490,23.360,154.117
C04336=1075.294,57.608,434.527,173.492,23.363,154.117
C04337=1075.300,57.857,434.509,173.493,23.366,154.117
C04338=1075.306,58.107,434.492,173.495,23.368,154.118
C04339=1075.312,58.356,434.476,173.496,23.370,154.118
C04340=1075.318,58.606,434.460,173.497,23.373,154.118
C04341=1075.323,58.855,434.443,173.499,23.376,154.119
C04342=1075.330,59.104,434.426,173.501,23.378,154.119
C04343=1075.336,59.353,434.410,173.502,23.381,154.119
C04344=1075.342,59.603,434.394,173.503,23.383,154.119
C04345=1075.347,59.852,434.377,173.505,23.386,154.120
C04346=1075.353,60.102,434.361,173.507,23.388,154.120
C04347=1075.360,60.351,434.343,173.508,23.391,154.120
C04348=1075.366,60.600,434.327,173.509,23.393,154.121
C04349=1075.371,60.850,434.310,173.511,23.396,154.121
C04350=1075.377,61.099,434.294,173.513,23.398,154.121
C04351=1075.383,61.348,434.277,173.514,23.401,154.121
C04352=1075.388,61.598,434.260,173.515,23.403,154.122
C04353=1075.394,61.847,434.244,173.517,23.406,154.122
C04354=1075.401,62.097,434.226,173.519,23.409,154.122
C04355=1075.406,62.346,434.210,173.520,23.411,154.123
C04356=1075.413,62.628,434.191,173.521,23.414,154.123
C04357=1075.420,62.909,434.172,173.523,23.417,154.123
C04358=1075.426,63.190,434.153,173.525,23.419,154.124
C04359=1075.433,63.471,434.135,173.527,23.422,154.124
C04360=1075.439,63.720,434.118,173.528,23.425,154.124
C04361=1075.445,63.970,434.100,173.529,23.427,154.124
C04362=1075.451,64.220,434.084,173.532,23.430,154.125
C04363=1075.457,64.468,434.067,173.533,23.433,154.125
C04364=1075.462,64.718,434.050,173.534,23.435,154.125
C04365=1075.469,64.967,434.033,173.535,23.438,154.126
C04366=1075.474,65.216,434.017,173.537,23.440,154.126
C04367=1075.480,65.466,434.000,173.539,23.443,154.126
C04368=1075.486,65.715,433.982,173.540,23.445,154.126
C04369=1075.492,65.965,433.966,173.541,23.448,154.127
C04370=1075.497,66.214,433.949,173.543,23.450,154.127
C04371=1075.503,66.463,433.932,173.545,23.453,154.127
C04372=1075.509,66.712,433.915,173.546,23.456,154.128
C04373=1075.515,66.962,433.898,173.547,23.458,154.128
C04374=1075.521,67.212,433.881,173.549,23.460,154.128
C04375=1075.526,67.461,433.864,173.551,23.463,154.129
C04376=1075.532,67.710,433.847,173.552,23.466,154.129
C04377=1075.538,67.959,433.830,173.553,23.468,154.129
C04378=1075.544,68.209,433.813,173.555,23.470,154.129
C04379=1075.550,68.458,433.796,173.556,23.473,154.130
C04380=1075.556,68.708,433.779,173.558,23.476,154.130
C04381=1075.561,68.957,433.762,173.559,23.479,154.130
C04382=1075.567,69.206,433.744,173.561,23.481,154.131
C04383=1075.573,69.456,433.728,173.562,23.483,154.131
C04384=1075.579,69.705,433.710,173.564,23.486,154.131
C04385=1075.585,69.954,433.694,173.565,23.488,154.132
C04386=1075.590,70.203,433.676,173.567,23.491,154.132
C04387=1075.595,70.453,433.659,173.568,23.494,154.132
C04388=1075.602,70.702,433.642,173.570,23.497,154.132
C04389=1075.607,70.952,433.625,173.571,23.499,154.133
C04390=1075.613,71.201,433.608,173.573,23.501,154.133
C04391=1075.618,71.450,433.590,173.574,23.504,154.133
C04392=1075.625,71.700,433.573,173.576,23.507,154.134
C04393=1075.631,71.949,433.556,173.578,23.509,154.134
C04394=1075.636,72.198,433.538,173.579,23.512,154.134
C04395=1075.642,72.448,433.522,173.580,23.514,154.135
C04396=1075.648,72.697,433.505,173.582,23.517,154.135
C04397=1075.654,72.946,433.487,173.583,23.519,154.135
C04398=1075.659,73.196,433.470,173.585,23.522,154.135
C04399=1075.665,73.445,433.453,173.586,23.524,154.136
C04400=1075.671,73.694,433.435,173.588,23.527,154.136
C04401=1075.676,73.944,433.418,173.590,23.529,154.136
C04402=1075.682,74.193,433.400,173.591,23.532,154.137
C04403=1075.688,74.442,433.383,173.592,23.535,154.137
C04404=1075.694,74.692,433.366,173.594,23.537,154.137
C04405=1075.700,74.941,433.349,173.596,23.540,154.138
C04406=1075.705,75.190,433.331,173.597,23.542,154.138
C04407=1075.711,75.439,433.314,173.598,23.545,154.138
C04408=1075.717,75.690,433.297,173.600,23.547,154.138
C04409=1075.723,75.939,433.279,173.602,23.550,154.139
C04410=1075.728,76.188,433.262,173.603,23.552,154.139
C04411=1075.735,76.437,433.244,173.604,23.555,154.139
C04412=1075.740,76.687,433.228,173.607,23.557,154.139
C04413=1075.746,76.936,433.210,173.608,23.560,154.140
C04414=1075.752,77.185,433.192,173.609,23.563,154.140
C04415=1075.757,77.434,433.175,173.611,23.565,154.140
C04416=1075.764,77.683,433.158,173.612,23.568,154.141
C04417=1075.769,77.934,433.140,173.614,23.570,154.141
C04418=1075.775,78.183,433.123,173.615,23.573,154.141
C04419=1075.781,78.432,433.105,173.617,23.575,154.142
C04420=1075.787,78.713,433.085,173.618,23.578,154.142
C04421=1075.794,78.994,433.065,173.621,23.581,154.142
C04422=1075.800,79.275,433.046,173.622,23.584,154.143
C04423=1075.806,79.556,433.026,173.624,23.587,154.143
C04424=1075.813,79.806,433.008,173.625,23.589,154.143
C04425=1075.818,80.055,432.990,173.627,23.592,154.143
C04426=1075.824,80.304,432.973,173.629,23.595,154.144
C04427=1075.829,80.553,432.955,173.630,23.597,154.144
C04428=1075.835,80.803,432.938,173.631,23.600,154.144
C04429=1075.840,81.052,432.921,173.633,23.602,154.145
C04430=1075.846,81.302,432.903,173.635,23.605,154.145
C04431=1075.852,81.551,432.885,173.636,23.607,154.145
C04432=1075.858,81.800,432.868,173.637,23.610,154.146
C04433=1075.864,82.050,432.850,173.640,23.612,154.146
C04434=1075.869,82.299,432.832,173.641,23.615,154.146
C04435=1075.875,82.548,432.814,173.642,23.618,154.147
C04436=1075.881,82.798,432.797,173.643,23.620,154.147
C04437=1075.886,83.047,432.779,173.646,23.623,154.147
C04438=1075.892,83.296,432.761,173.647,23.625,154.147
C04439=1075.898,83.546,432.743,173.648,23.628,154.148
C04440=1075.904,83.795,432.726,173.650,23.630,154.148
C04441=1075.909,84.044,432.708,173.652,23.633,154.148
C04442=1075.915,84.294,432.690,173.653,23.635,154.148
C04443=1075.921,84.543,432.673,173.654,23.638,154.149
C04444=1075.927,84.792,432.655,173.657,23.640,154.149
C04445=1075.932,85.041,432.637,173.658,23.643,154.149
C04446=1075.939,85.290,432.619,173.659,23.645,154.150
C04447=1075.944,85.539,432.601,173.660,23.648,154.150
C04448=1075.950,85.789,432.584,173.663,23.651,154.150
C04449=1075.955,86.039,432.565,173.664,23.653,154.151
C04450=1075.961,86.288,432.547,173.665,23.655,154.151
C04451=1075.967,86.537,432.529,173.668,23.658,154.151
C04452=1075.972,86.786,432.512,173.669,23.661,154.151
C04453=1075.979,87.036,432.494,173.670,23.663,154.152
C04454=1075.984,87.285,432.476,173.671,23.665,154.152
C04455=1075.990,87.534,432.458,173.674,23.668,154.152
C04456=1075.996,87.783,432.440,173.675,23.671,154.153
C04457=1076.002,88.032,432.423,173.676,23.673,154.153
C04458=1076.008,88.282,432.405,173.679,23.676,154.153
C04459=1076.013,88.531,432.387,173.680,23.678,154.153
C04460=1076.019,88.781,432.369,173.681,23.680,154.154
C04461=1076.025,89.029,432.351,173.683,23.683,154.154
C04462=1076.030,89.279,432.332,173.685,23.686,154.154
C04463=1076.036,89.528,432.315,173.686,23.688,154.155
C04464=1076.042,89.778,432.297,173.687,23.690,154.155
C04465=1076.048,90.027,432.279,173.690,23.693,154.155
C04466=1076.054,90.276,432.261,173.691,23.696,154.155
C04467=1076.060,90.525,432.243,173.692,23.698,154.156
C04468=1076.066,90.775,432.225,173.694,23.701,154.156
C04469=1076.072,91.024,432.207,173.696,23.703,154.156
C04470=1076.077,91.274,432.188,173.697,23.705,154.156
C04471=1076.082,91.523,432.171,173.699,23.708,154.157
C04472=1076.089,91.772,432.153,173.701,23.711,154.157
C04473=1076.094,92.021,432.134,173.702,23.713,154.157
C04474=1076.100,92.271,432.116,173.704,23.716,154.158
C04475=1076.105,92.520,432.099,173.705,23.718,154.158
C04476=1076.111,92.769,432.079,173.707,23.721,154.158
C04477=1076.116,93.018,432.062,173.708,23.723,154.159
C04478=1076.123,93.268,432.044,173.710,23.726,154.159
C04479=1076.128,93.517,432.025,173.711,23.728,154.159
C04480=1076.134,93.767,432.007,173.713,23.731,154.159
C04481=1076.139,94.016,431.989,173.715,23.734,154.160
C04482=1076.146,94.265,431.971,173.716,23.736,154.160
C04483=1076.151,94.514,431.953,173.718,23.738,154.160
C04484=1076.157,94.796,431.932,173.720,23.741,154.161
C04485=1076.164,95.076,431.911,173.722,23.744,154.161
C04486=1076.170,95.358,431.890,173.723,23.747,154.161
C04487=1076.177,95.639,431.870,173.725,23.750,154.162
C04488=1076.183,95.888,431.852,173.727,23.752,154.162
C04489=1076.188,96.138,431.833,173.728,23.755,154.162
C04490=1076.194,96.386,431.815,173.730,23.758,154.162
C04491=1076.200,96.636,431.797,173.732,23.760,154.163
C04492=1076.205,96.885,431.778,173.733,23.762,154.163
C04493=1076.211,97.135,431.760,173.735,23.765,154.163
C04494=1076.218,97.384,431.742,173.736,23.767,154.164
C04495=1076.222,97.633,431.723,173.738,23.770,154.164
C04496=1076.229,97.882,431.705,173.740,23.773,154.164
C04497=1076.234,98.131,431.687,173.741,23.775,154.164
C04498=1076.240,98.381,431.668,173.743,23.777,154.165
C04499=1076.246,98.630,431.650,173.745,23.780,154.165
C04500=1076.251,98.879,431.631,173.746,23.782,154.165
C04501=1076.257,99.129,431.613,173.748,23.784,154.165
C04502=1076.262,99.378,431.594,173.750,23.787,154.166
C04503=1076.269,99.627,431.576,173.751,23.789,154.166
C04504=1076.275,99.876,431.558,173.753,23.792,154.166
C04505=1076.280,100.126,431.540,173.755,23.795,154.166
C04506=1076.286,100.375,431.521,173.756,23.797,154.167
C04507=1076.292,100.624,431.502,173.757,23.799,154.167
C04508=1076.297,100.873,431.484,173.760,23.802,154.167
C04509=1076.304,101.122,431.465,173.761,23.804,154.168
C04510=1076.309,101.371,431.447,173.762,23.807,154.168
C04511=1076.315,101.621,431.429,173.764,23.810,154.168
C04512=1076.321,101.870,431.409,173.766,23.812,154.168
C04513=1076.325,102.120,431.391,173.767,23.814,154.169
C04514=1076.332,102.369,431.373,173.769,23.817,154.169
C04515=1076.337,102.618,431.354,173.771,23.819,154.169
C04516=1076.343,102.867,431.336,173.772,23.822,154.170
C04517=1076.349,103.117,431.317,173.774,23.825,154.170
C04518=1076.354,103.366,431.298,173.776,23.827,154.170
C04519=1076.360,103.615,431.279,173.778,23.830,154.170
C04520=1076.366,103.865,431.260,173.779,23.832,154.171
C04521=1076.371,104.113,431.242,173.780,23.834,154.171
C04522=1076.377,104.363,431.223,173.783,23.837,154.171
C04523=1076.383,104.613,431.204,173.784,23.840,154.172
C04524=1076.388,104.861,431.186,173.785,23.842,154.172
C04525=1076.394,105.110,431.167,173.788,23.845,154.172
C04526=1076.400,105.360,431.148,173.789,23.847,154.172
C04527=1076.406,105.608,431.129,173.790,23.849,154.173
C04528=1076.411,105.858,431.111,173.792,23.852,154.173
C04529=1076.417,106.108,431.092,173.794,23.855,154.173
C04530=1076.423,106.356,431.073,173.795,23.857,154.173
C04531=1076.428,106.606,431.054,173.797,23.860,154.174
C04532=1076.434,106.855,431.035,173.799,23.862,154.174
C04533=1076.439,107.104,431.017,173.801,23.865,154.174
C04534=1076.445,107.354,430.998,173.802,23.867,154.175
C04535=1076.451,107.603,430.979,173.804,23.869,154.175
C04536=1076.457,107.852,430.960,173.806,23.872,154.175
C04537=1076.462,108.101,430.941,173.807,23.875,154.175
C04538=1076.468,108.350,430.922,173.809,23.877,154.176
C04539=1076.474,108.599,430.903,173.811,23.879,154.176
C04540=1076.480,108.849,430.885,173.812,23.882,154.176
C04541=1076.485,109.098,430.866,173.814,23.884,154.176
C04542=1076.491,109.347,430.847,173.816,23.887,154.177
C04543=1076.497,109.597,430.828,173.817,23.889,154.177
C04544=1076.503,109.846,430.809,173.819,23.892,154.177
C04545=1076.508,110.095,430.791,173.821,23.894,154.178
C04546=1076.514,110.344,430.771,173.822,23.896,154.178
C04547=1076.520,110.593,430.752,173.824,23.899,154.178
C04548=1076.527,110.874,430.731,173.826,23.902,154.178
C04549=1076.533,111.156,430.709,173.828,23.904,154.179
C04550=1076.539,111.438,430.688,173.830,23.907,154.179
C04551=1076.546,111.719,430.667,173.832,23.910,154.179
C04552=1076.551,111.968,430.648,173.834,23.913,154.180
C04553=1076.557,112.217,430.629,173.835,23.915,154.180
C04554=1076.563,112.466,430.610,173.837,23.918,154.180
C04555=1076.569,112.716,430.590,173.839,23.920,154.180
C04556=1076.574,112.964,430.572,173.840,23.922,154.181
C04557=1076.580,113.214,430.552,173.842,23.925,154.181
C04558=1076.585,113.463,430.533,173.843,23.927,154.181
C04559=1076.592,113.712,430.514,173.846,23.930,154.181
C04560=1076.598,113.961,430.495,173.847,23.932,154.182
C04561=1076.603,114.210,430.476,173.848,23.935,154.182
C04562=1076.608,114.459,430.456,173.851,23.937,154.182
C04563=1076.614,114.709,430.437,173.852,23.940,154.183
C04564=1076.620,114.958,430.418,173.854,23.942,154.183
C04565=1076.626,115.208,430.399,173.856,23.945,154.183
C04566=1076.631,115.456,430.380,173.857,23.947,154.183
C04567=1076.636,115.706,430.361,173.859,23.950,154.184
C04568=1076.642,115.955,430.341,173.860,23.952,154.184
C04569=1076.648,116.204,430.321,173.863,23.955,154.184
C04570=1076.653,116.453,430.302,173.864,23.957,154.184
C04571=1076.659,116.702,430.283,173.865,23.960,154.185
C04572=1076.664,116.952,430.264,173.868,23.962,154.185
C04573=1076.670,117.201,430.245,173.869,23.965,154.185
C04574=1076.676,117.450,430.225,173.871,23.968,154.186
C04575=1076.681,117.699,430.206,173.873,23.969,154.186
C04576=1076.687,117.948,430.187,173.874,23.972,154.186
C04577=1076.693,118.197,430.167,173.876,23.974,154.186
C04578=1076.698,118.447,430.148,173.878,23.977,154.187
C04579=1076.704,118.696,430.128,173.880,23.980,154.187
C04580=1076.709,118.945,430.108,173.881,23.982,154.187
C04581=1076.714,119.194,430.090,173.883,23.985,154.187
C04582=1076.720,119.443,430.070,173.885,23.987,154.188
C04583=1076.726,119.692,430.050,173.886,23.989,154.188
C04584=1076.732,119.942,430.031,173.888,23.992,154.188
C04585=1076.737,120.191,430.012,173.890,23.994,154.189
C04586=1076.743,120.440,429.992,173.892,23.997,154.189
C04587=1076.749,120.690,429.973,173.893,24.000,154.189
C04588=1076.754,120.938,429.954,173.895,24.001,154.189
C04589=1076.760,121.187,429.934,173.897,24.004,154.189
C04590=1076.765,121.437,429.914,173.898,24.006,154.190
C04591=1076.771,121.686,429.895,173.901,24.009,154.190
C04592=1076.777,121.935,429.875,173.902,24.012,154.190
C04593=1076.782,122.184,429.855,173.904,24.014,154.191
C04594=1076.788,122.434,429.836,173.906,24.017,154.191
C04595=1076.794,122.683,429.816,173.907,24.019,154.191
C04596=1076.800,122.932,429.797,173.909,24.021,154.191
C04597=1076.806,123.181,429.777,173.911,24.024,154.192
C04598=1076.810,123.430,429.758,173.913,24.026,154.192
C04599=1076.816,123.679,429.738,173.914,24.029,154.192
C04600=1076.822,123.928,429.718,173.917,24.031,154.192
C04601=1076.828,124.178,429.699,173.918,24.034,154.193
C04602=1076.833,124.427,429.679,173.920,24.036,154.193
C04603=1076.839,124.676,429.660,173.922,24.038,154.193
C04604=1076.845,124.925,429.640,173.923,24.041,154.193
C04605=1076.850,125.175,429.620,173.925,24.043,154.194
C04606=1076.856,125.423,429.600,173.927,24.046,154.194
C04607=1076.862,125.673,429.581,173.929,24.048,154.194
C04608=1076.868,125.922,429.561,173.930,24.050,154.194
C04609=1076.873,126.171,429.542,173.933,24.053,154.195
C04610=1076.879,126.420,429.522,173.934,24.055,154.195
C04611=1076.885,126.669,429.503,173.936,24.058,154.195
C04612=1076.891,126.950,429.480,173.937,24.060,154.196
C04613=1076.898,127.231,429.458,173.940,24.063,154.196
C04614=1076.905,127.513,429.435,173.942,24.066,154.196
C04615=1076.910,127.794,429.413,173.944,24.069,154.196
C04616=1076.916,128.043,429.393,173.946,24.071,154.197
C04617=1076.922,128.293,429.374,173.948,24.074,154.197
C04618=1076.928,128.542,429.354,173.949,24.076,154.197
C04619=1076.934,128.790,429.334,173.952,24.078,154.197
C04620=1076.939,129.040,429.314,173.953,24.081,154.198
C04621=1076.945,129.289,429.294,173.954,24.083,154.198
C04622=1076.951,129.538,429.274,173.957,24.086,154.198
C04623=1076.957,129.787,429.255,173.958,24.088,154.198
C04624=1076.963,130.036,429.235,173.960,24.090,154.199
C04625=1076.968,130.286,429.215,173.962,24.093,154.199
C04626=1076.974,130.535,429.194,173.964,24.095,154.199
C04627=1076.980,130.784,429.175,173.965,24.097,154.199
C04628=1076.986,131.033,429.155,173.968,24.100,154.199
C04629=1076.991,131.283,429.135,173.969,24.102,154.200
C04630=1076.997,131.531,429.115,173.971,24.104,154.200
C04631=1077.003,131.780,429.095,173.973,24.107,154.200
C04632=1077.009,132.030,429.076,173.975,24.109,154.200
C04633=1077.014,132.279,429.055,173.976,24.112,154.201
C04634=1077.020,132.528,429.035,173.979,24.115,154.201
C04635=1077.025,132.777,429.015,173.980,24.116,154.201
C04636=1077.031,133.026,428.995,173.982,24.119,154.201
C04637=1077.037,133.275,428.975,173.984,24.121,154.202
C04638=1077.042,133.524,428.955,173.986,24.124,154.202
C04639=1077.049,133.774,428.934,173.987,24.127,154.202
C04640=1077.054,134.023,428.914,173.990,24.129,154.202
C04641=1077.060,134.272,428.895,173.991,24.131,154.203
C04642=1077.065,134.521,428.874,173.993,24.134,154.203
C04643=1077.071,134.770,428.854,173.995,24.136,154.203
C04644=1077.076,135.019,428.834,173.997,24.139,154.204
C04645=1077.082,135.268,428.814,173.998,24.141,154.204
C04646=1077.088,135.517,428.793,174.001,24.143,154.204
C04647=1077.094,135.766,428.773,174.002,24.146,154.204
C04648=1077.099,136.016,428.753,174.004,24.148,154.205
C04649=1077.105,136.265,428.733,174.006,24.150,154.205
C04650=1077.110,136.514,428.712,174.008,24.153,154.205
C04651=1077.116,136.763,428.692,174.009,24.155,154.205
C04652=1077.122,137.012,428.672,174.012,24.158,154.206
C04653=1077.128,137.261,428.652,174.013,24.160,154.206
C04654=1077.133,137.510,428.631,174.016,24.163,154.206
C04655=1077.139,137.759,428.611,174.017,24.165,154.206
C04656=1077.144,138.008,428.591,174.019,24.168,154.206
C04657=1077.151,138.258,428.571,174.021,24.169,154.207
C04658=1077.156,138.507,428.550,174.023,24.172,154.207
C04659=1077.162,138.756,428.530,174.024,24.175,154.207
C04660=1077.167,139.005,428.509,174.027,24.177,154.207
C04661=1077.173,139.254,428.489,174.028,24.179,154.208
C04662=1077.179,139.503,428.469,174.030,24.182,154.208
C04663=1077.184,139.752,428.448,174.032,24.184,154.208
C04664=1077.190,140.001,428.428,174.034,24.187,154.208
C04665=1077.196,140.250,428.407,174.035,24.189,154.209
C04666=1077.202,140.499,428.388,174.038,24.191,154.209
C04667=1077.207,140.748,428.367,174.039,24.194,154.209
C04668=1077.212,140.997,428.346,174.041,24.196,154.209
C04669=1077.218,141.247,428.326,174.043,24.199,154.210
C04670=1077.224,141.496,428.306,174.045,24.201,154.210
C04671=1077.229,141.745,428.285,174.047,24.204,154.210
C04672=1077.235,141.994,428.264,174.049,24.206,154.210
C04673=1077.241,142.243,428.244,174.051,24.209,154.211
C04674=1077.247,142.492,428.223,174.052,24.211,154.211
C04675=1077.252,142.742,428.202,174.055,24.213,154.211
C04676=1077.258,143.022,428.179,174.057,24.216,154.211
C04677=1077.264,143.304,428.156,174.058,24.218,154.212
C04678=1077.271,143.585,428.133,174.061,24.221,154.212
C04679=1077.277,143.865,428.110,174.063,24.224,154.212
C04680=1077.283,144.115,428.089,174.065,24.226,154.212
C04681=1077.289,144.364,428.068,174.066,24.229,154.213
C04682=1077.294,144.613,428.048,174.069,24.231,154.213
C04683=1077.300,144.862,428.028,174.070,24.233,154.213
C04684=1077.306,145.111,428.006,174.073,24.236,154.213
C04685=1077.311,145.360,427.986,174.075,24.239,154.214
C04686=1077.317,145.610,427.965,174.076,24.241,154.214
C04687=1077.322,145.858,427.945,174.079,24.243,154.214
C04688=1077.329,146.108,427.923,174.080,24.246,154.214
C04689=1077.334,146.357,427.903,174.082,24.248,154.215
C04690=1077.339,146.606,427.882,174.084,24.250,154.215
C04691=1077.345,146.855,427.862,174.086,24.253,154.215
C04692=1077.351,147.104,427.841,174.087,24.255,154.215
C04693=1077.357,147.353,427.820,174.090,24.257,154.216
C04694=1077.362,147.602,427.800,174.092,24.260,154.216
C04695=1077.368,147.851,427.778,174.093,24.262,154.216
C04696=1077.374,148.100,427.758,174.096,24.265,154.216
C04697=1077.379,148.349,427.737,174.097,24.267,154.217
C04698=1077.385,148.598,427.716,174.099,24.270,154.217
C04699=1077.391,148.848,427.695,174.101,24.272,154.217
C04700=1077.396,149.096,427.674,174.103,24.274,154.217
C04701=1077.401,149.345,427.653,174.106,24.277,154.217
C04702=1077.407,149.595,427.633,174.107,24.279,154.218
C04703=1077.413,149.843,427.611,174.109,24.281,154.218
C04704=1077.418,150.093,427.591,174.111,24.284,154.218
C04705=1077.424,150.342,427.569,174.113,24.286,154.218
C04706=1077.430,150.591,427.548,174.115,24.289,154.219
C04707=1077.436,150.839,427.528,174.117,24.291,154.219
C04708=1077.442,151.089,427.507,174.119,24.294,154.219
C04709=1077.447,151.338,427.486,174.120,24.296,154.219
C04710=1077.453,151.587,427.465,174.123,24.298,154.220
C04711=1077.458,151.836,427.444,174.125,24.301,154.220
C04712=1077.464,152.085,427.423,174.126,24.303,154.220
C04713=1077.469,152.334,427.402,174.129,24.306,154.220
C04714=1077.475,152.583,427.381,174.130,24.308,154.221
C04715=1077.481,152.832,427.360,174.132,24.310,154.221
C04716=1077.486,153.081,427.339,174.135,24.313,154.221
C04717=1077.492,153.330,427.317,174.136,24.315,154.221
C04718=1077.498,153.579,427.297,174.139,24.318,154.222
C04719=1077.503,153.828,427.275,174.140,24.320,154.222
C04720=1077.508,154.078,427.254,174.142,24.322,154.222
C04721=1077.514,154.326,427.233,174.145,24.325,154.222
C04722=1077.520,154.576,427.212,174.146,24.327,154.223
C04723=1077.525,154.825,427.190,174.148,24.329,154.223
C04724=1077.531,155.073,427.169,174.150,24.332,154.223
C04725=1077.537,155.323,427.148,174.152,24.334,154.223
C04726=1077.542,155.572,427.127,174.154,24.337,154.223
C04727=1077.548,155.821,427.105,174.156,24.339,154.224
C04728=1077.554,156.070,427.085,174.158,24.342,154.224
C04729=1077.559,156.318,427.064,174.160,24.344,154.224
C04730=1077.565,156.568,427.042,174.162,24.346,154.224
C04731=1077.571,156.817,427.021,174.164,24.349,154.225
C04732=1077.576,157.066,426.999,174.166,24.351,154.225
C04733=1077.582,157.315,426.978,174.168,24.353,154.225
C04734=1077.588,157.565,426.957,174.170,24.356,154.225
C04735=1077.593,157.813,426.936,174.172,24.358,154.226
C04736=1077.599,158.062,426.914,174.174,24.360,154.226
C04737=1077.605,158.311,426.893,174.176,24.363,154.226
C04738=1077.609,158.560,426.872,174.178,24.365,154.226
C04739=1077.615,158.809,426.850,174.180,24.368,154.226
C04740=1077.622,159.090,426.826,174.182,24.370,154.227
C04741=1077.629,159.371,426.802,174.185,24.373,154.227
C04742=1077.634,159.651,426.778,174.187,24.376,154.227
C04743=1077.641,159.933,426.754,174.189,24.378,154.227
C04744=1077.647,160.182,426.732,174.191,24.381,154.228
C04745=1077.653,160.430,426.711,174.193,24.383,154.228
C04746=1077.658,160.680,426.689,174.195,24.386,154.228
C04747=1077.663,160.929,426.668,174.197,24.388,154.228
C04748=1077.670,161.178,426.646,174.199,24.390,154.229
C04749=1077.675,161.427,426.625,174.201,24.393,154.229
C04750=1077.680,161.675,426.603,174.203,24.395,154.229
C04751=1077.686,161.925,426.582,174.205,24.398,154.229
C04752=1077.691,162.173,426.560,174.207,24.400,154.230
C04753=1077.697,162.423,426.538,174.209,24.402,154.230
C04754=1077.702,162.671,426.516,174.211,24.405,154.230
C04755=1077.708,162.921,426.495,174.213,24.408,154.230
C04756=1077.713,163.169,426.473,174.215,24.410,154.231
C04757=1077.719,163.418,426.451,174.217,24.412,154.231
C04758=1077.724,163.667,426.429,174.219,24.415,154.231
C04759=1077.729,163.916,426.408,174.221,24.417,154.231
C04760=1077.735,164.165,426.386,174.223,24.420,154.232
C04761=1077.740,164.415,426.365,174.226,24.422,154.232
C04762=1077.746,164.664,426.342,174.227,24.424,154.232
C04763=1077.751,164.912,426.321,174.229,24.427,154.232
C04764=1077.757,165.162,426.299,174.231,24.430,154.233
C04765=1077.762,165.410,426.277,174.233,24.432,154.233
C04766=1077.768,165.660,426.255,174.235,24.434,154.233
C04767=1077.773,165.908,426.234,174.238,24.437,154.233
C04768=1077.779,166.158,426.212,174.240,24.440,154.234
C04769=1077.784,166.406,426.190,174.241,24.442,154.234
C04770=1077.790,166.656,426.168,174.244,24.444,154.234
C04771=1077.795,166.904,426.147,174.246,24.447,154.234
C04772=1077.801,167.154,426.125,174.247,24.449,154.235
C04773=1077.806,167.402,426.103,174.250,24.451,154.235
C04774=1077.812,167.652,426.081,174.252,24.454,154.235
C04775=1077.817,167.900,426.059,174.253,24.456,154.235
C04776=1077.823,168.149,426.037,174.256,24.459,154.235
C04777=1077.829,168.399,426.015,174.258,24.461,154.236
C04778=1077.834,168.647,425.994,174.260,24.464,154.236
C04779=1077.840,168.897,425.971,174.262,24.466,154.236
C04780=1077.845,169.145,425.950,174.264,24.468,154.236
C04781=1077.851,169.394,425.927,174.267,24.471,154.237
C04782=1077.856,169.643,425.905,174.268,24.473,154.237
C04783=1077.862,169.892,425.884,174.270,24.476,154.237
C04784=1077.867,170.142,425.861,174.273,24.478,154.237
C04785=1077.873,170.390,425.840,174.275,24.481,154.238
C04786=1077.879,170.639,425.817,174.276,24.483,154.238
C04787=1077.884,170.888,425.795,174.279,24.485,154.238
C04788=1077.890,171.137,425.774,174.281,24.488,154.238
C04789=1077.895,171.386,425.751,174.282,24.490,154.239
C04790=1077.901,171.634,425.729,174.285,24.493,154.239
C04791=1077.906,171.884,425.707,174.287,24.495,154.239
C04792=1077.912,172.133,425.685,174.290,24.497,154.239
C04793=1077.918,172.381,425.663,174.291,24.500,154.239
C04794=1077.923,172.631,425.641,174.293,24.502,154.240
C04795=1077.929,172.880,425.619,174.296,24.505,154.240
C04796=1077.934,173.128,425.597,174.298,24.507,154.240
C04797=1077.940,173.378,425.574,174.299,24.510,154.240
C04798=1077.946,173.627,425.553,174.302,24.512,154.240
C04799=1077.951,173.875,425.530,174.304,24.514,154.241
C04800=1077.956,174.125,425.508,174.306,24.517,154.241
C04801=1077.963,174.373,425.485,174.308,24.519,154.241
C04802=1077.968,174.622,425.464,174.310,24.522,154.241
C04803=1077.973,174.871,425.441,174.313,24.524,154.242
C04804=1077.980,175.152,425.417,174.315,24.526,154.242
C04805=1077.987,175.433,425.391,174.317,24.529,154.242
C04806=1077.993,175.713,425.366,174.319,24.532,154.242
C04807=1077.999,175.993,425.341,174.322,24.535,154.243
C04808=1078.005,176.242,425.318,174.324,24.537,154.243
C04809=1078.010,176.491,425.296,174.327,24.539,154.243
C04810=1078.016,176.740,425.274,174.329,24.542,154.243
C04811=1078.022,176.989,425.252,174.330,24.544,154.244
C04812=1078.028,177.238,425.229,174.333,24.547,154.244
C04813=1078.033,177.487,425.207,174.335,24.549,154.244
C04814=1078.038,177.736,425.184,174.337,24.551,154.244
C04815=1078.045,177.985,425.163,174.340,24.554,154.244
C04816=1078.050,178.234,425.140,174.341,24.556,154.245
C04817=1078.056,178.483,425.117,174.343,24.559,154.245
C04818=1078.062,178.731,425.095,174.346,24.561,154.245
C04819=1078.067,178.981,425.073,174.348,24.563,154.245
C04820=1078.073,179.229,425.050,174.350,24.566,154.246
C04821=1078.079,179.478,425.027,174.352,24.568,154.246
C04822=1078.085,179.728,425.006,174.354,24.571,154.246
C04823=1078.090,179.976,424.983,174.357,24.573,154.246
C04824=1078.096,180.225,424.960,174.359,24.575,154.246
C04825=1078.102,180.474,424.938,174.360,24.578,154.247
C04826=1078.107,180.723,424.915,174.363,24.580,154.247
C04827=1078.113,180.972,424.893,174.365,24.582,154.247
C04828=1078.119,181.221,424.870,174.368,24.585,154.247
C04829=1078.125,181.470,424.848,174.370,24.587,154.247
C04830=1078.130,181.718,424.825,174.371,24.589,154.248
C04831=1078.136,181.968,424.803,174.374,24.592,154.248
C04832=1078.141,182.216,424.780,174.376,24.594,154.248
C04833=1078.147,182.465,424.757,174.379,24.597,154.248
C04834=1078.154,182.714,424.735,174.381,24.599,154.248
C04835=1078.159,182.963,424.713,174.383,24.601,154.249
C04836=1078.165,183.212,424.690,174.385,24.603,154.249
C04837=1078.170,183.461,424.667,174.387,24.606,154.249
C04838=1078.177,183.710,424.644,174.390,24.608,154.249
C04839=1078.183,183.959,424.621,174.392,24.611,154.250
C04840=1078.188,184.208,424.599,174.394,24.613,154.250
C04841=1078.193,184.456,424.577,174.397,24.616,154.250
C04842=1078.199,184.705,424.554,174.398,24.617,154.250
C04843=1078.205,184.954,424.531,174.400,24.620,154.250
C04844=1078.210,185.203,424.508,174.403,24.623,154.251
C04845=1078.216,185.452,424.485,174.405,24.625,154.251
C04846=1078.222,185.701,424.462,174.407,24.627,154.251
C04847=1078.227,185.950,424.440,174.410,24.630,154.251
C04848=1078.232,186.199,424.417,174.411,24.632,154.252
C04849=1078.237,186.448,424.394,174.413,24.635,154.252
C04850=1078.243,186.697,424.371,174.416,24.637,154.252
C04851=1078.249,186.946,424.348,174.418,24.640,154.252
C04852=1078.255,187.194,424.325,174.420,24.643,154.253
C04853=1078.260,187.443,424.302,174.423,24.645,154.253
C04854=1078.266,187.692,424.279,174.424,24.647,154.253
C04855=1078.270,187.941,424.256,174.427,24.650,154.253
C04856=1078.276,188.190,424.233,174.429,24.652,154.254
C04857=1078.282,188.439,424.210,174.431,24.655,154.254
C04858=1078.288,188.687,424.187,174.434,24.657,154.254
C04859=1078.293,188.937,424.163,174.436,24.660,154.254
C04860=1078.298,189.186,424.140,174.438,24.663,154.254
C04861=1078.304,189.434,424.117,174.440,24.664,154.255
C04862=1078.310,189.683,424.094,174.442,24.667,154.255
C04863=1078.316,189.932,424.072,174.444,24.670,154.255
C04864=1078.320,190.181,424.048,174.447,24.672,154.255
C04865=1078.326,190.430,424.025,174.449,24.675,154.256
C04866=1078.332,190.678,424.002,174.451,24.677,154.256
C04867=1078.337,190.927,423.979,174.454,24.680,154.256
C04868=1078.343,191.208,423.953,174.456,24.683,154.256
C04869=1078.350,191.488,423.927,174.458,24.685,154.257
C04870=1078.355,191.768,423.900,174.462,24.688,154.257
C04871=1078.362,192.048,423.874,174.464,24.691,154.257
C04872=1078.368,192.297,423.851,174.466,24.693,154.257
C04873=1078.374,192.546,423.828,174.469,24.696,154.258
C04874=1078.379,192.795,423.805,174.470,24.698,154.258
C04875=1078.385,193.043,423.781,174.473,24.700,154.258
C04876=1078.390,193.292,423.758,174.475,24.703,154.258
C04877=1078.395,193.541,423.735,174.477,24.706,154.259
C04878=1078.401,193.790,423.712,174.480,24.708,154.259
C04879=1078.407,194.038,423.688,174.482,24.710,154.259
C04880=1078.413,194.287,423.665,174.484,24.713,154.259
C04881=1078.418,194.537,423.642,174.486,24.716,154.259
C04882=1078.424,194.785,423.619,174.489,24.718,154.260
C04883=1078.430,195.034,423.595,174.491,24.720,154.260
C04884=1078.435,195.283,423.571,174.494,24.723,154.260
C04885=1078.440,195.532,423.548,174.495,24.725,154.260
C04886=1078.446,195.780,423.525,174.497,24.728,154.261
C04887=1078.452,196.030,423.501,174.500,24.730,154.261
C04888=1078.458,196.279,423.478,174.502,24.732,154.261
C04889=1078.464,196.527,423.454,174.504,24.735,154.261
C04890=1078.469,196.776,423.431,174.507,24.737,154.261
C04891=1078.474,197.025,423.408,174.509,24.740,154.262
C04892=1078.480,197.274,423.384,174.512,24.743,154.262
C04893=1078.485,197.523,423.361,174.514,24.745,154.262
C04894=1078.491,197.771,423.337,174.516,24.747,154.262
C04895=1078.497,198.020,423.314,174.519,24.750,154.263
C04896=1078.502,198.269,423.290,174.521,24.752,154.263
C04897=1078.509,198.518,423.266,174.523,24.755,154.263
C04898=1078.514,198.767,423.243,174.526,24.757,154.263
C04899=1078.520,199.016,423.219,174.528,24.760,154.263
C04900=1078.526,199.264,423.196,174.530,24.762,154.264
C04901=1078.531,199.513,423.172,174.533,24.764,154.264
C04902=1078.537,199.762,423.149,174.534,24.767,154.264
C04903=1078.543,200.011,423.125,174.537,24.769,154.264
C04904=1078.548,200.260,423.101,174.539,24.771,154.265
C04905=1078.554,200.508,423.078,174.541,24.774,154.265
C04906=1078.559,200.758,423.054,174.544,24.777,154.265
C04907=1078.565,201.006,423.031,174.546,24.779,154.265
C04908=1078.571,201.254,423.007,174.548,24.782,154.266
C04909=1078.577,201.504,422.983,174.551,24.784,154.266
C04910=1078.583,201.752,422.959,174.553,24.786,154.266
C04911=1078.588,202.002,422.936,174.556,24.789,154.266
C04912=1078.594,202.250,422.912,174.558,24.791,154.266
C04913=1078.600,202.499,422.888,174.560,24.794,154.267
C04914=1078.606,202.748,422.865,174.563,24.796,154.267
C04915=1078.611,202.997,422.840,174.565,24.799,154.267
C04916=1078.617,203.245,422.817,174.567,24.801,154.267
C04917=1078.622,203.494,422.793,174.570,24.804,154.268
C04918=1078.627,203.743,422.769,174.572,24.807,154.268
C04919=1078.634,203.992,422.745,174.574,24.809,154.268
C04920=1078.639,204.241,422.721,174.577,24.811,154.268
C04921=1078.644,204.489,422.697,174.579,24.814,154.268
C04922=1078.650,204.738,422.673,174.581,24.817,154.269
C04923=1078.656,204.986,422.649,174.584,24.819,154.269
C04924=1078.661,205.236,422.625,174.586,24.821,154.269
C04925=1078.667,205.485,422.602,174.589,24.824,154.269
C04926=1078.672,205.733,422.577,174.591,24.827,154.270
C04927=1078.678,205.982,422.553,174.593,24.829,154.270
C04928=1078.683,206.231,422.530,174.596,24.832,154.270
C04929=1078.689,206.480,422.505,174.598,24.834,154.270
C04930=1078.695,206.728,422.481,174.600,24.837,154.271
C04931=1078.700,206.977,422.457,174.603,24.839,154.271
C04932=1078.724,208.013,422.357,174.708,24.895,154.270
C04933=1078.733,208.415,422.317,174.712,24.901,154.270
C04934=1078.742,208.817,422.277,174.715,24.906,154.271
C04935=1078.751,209.221,422.238,174.720,24.913,154.272
C04936=1078.761,209.623,422.197,174.723,24.918,154.273
C04937=1078.767,209.873,422.173,174.725,24.921,154.273
C04938=1078.772,210.120,422.148,174.727,24.925,154.274
C04939=1078.778,210.370,422.123,174.730,24.928,154.274
C04940=1078.784,210.618,422.098,174.732,24.932,154.275
C04941=1078.790,210.867,422.074,174.734,24.935,154.275
C04942=1078.795,211.116,422.049,174.736,24.939,154.275
C04943=1078.801,211.364,422.024,174.739,24.942,154.276
C04944=1078.806,211.613,422.000,174.741,24.946,154.276
C04945=1078.813,211.862,421.974,174.743,24.949,154.277
C04946=1078.818,212.110,421.950,174.745,24.953,154.277
C04947=1078.824,212.359,421.925,174.747,24.956,154.278
C04948=1078.829,212.607,421.901,174.749,24.960,154.278
C04949=1078.835,212.856,421.875,174.753,24.963,154.279
C04950=1078.841,213.106,421.850,174.755,24.967,154.279
C04951=1078.846,213.354,421.825,174.757,24.970,154.279
C04952=1078.852,213.603,421.800,174.759,24.974,154.280
C04953=1078.858,213.851,421.775,174.761,24.977,154.280
C04954=1078.863,214.100,421.750,174.763,24.981,154.281
C04955=1078.869,214.348,421.725,174.765,24.984,154.281
C04956=1078.875,214.597,421.700,174.768,24.988,154.282
C04957=1078.881,214.846,421.675,174.770,24.991,154.282
C04958=1078.886,215.094,421.650,174.772,24.995,154.283
C04959=1078.892,215.344,421.625,174.774,24.998,154.283
C04960=1078.897,215.592,421.600,174.777,25.001,154.284
C04961=1078.903,215.841,421.575,174.780,25.005,154.284
C04962=1078.909,216.090,421.550,174.782,25.009,154.285
C04963=1078.914,216.338,421.525,174.784,25.012,154.285
C04964=1078.920,216.587,421.499,174.786,25.015,154.286
C04965=1078.926,216.835,421.475,174.788,25.019,154.286
C04966=1078.931,217.084,421.449,174.790,25.022,154.286
C04967=1078.937,217.333,421.424,174.793,25.026,154.287
C04968=1078.943,217.581,421.399,174.795,25.029,154.287
C04969=1078.949,217.830,421.374,174.798,25.033,154.288
C04970=1078.954,218.079,421.348,174.800,25.036,154.288
C04971=1078.960,218.327,421.323,174.802,25.039,154.289
C04972=1078.966,218.576,421.298,174.805,25.044,154.289
C04973=1078.972,218.825,421.272,174.807,25.047,154.290
C04974=1078.977,219.074,421.248,174.809,25.050,154.290
C04975=1078.983,219.322,421.222,174.811,25.054,154.290
C04976=1078.989,219.571,421.197,174.813,25.057,154.291
C04977=1078.995,219.820,421.171,174.816,25.061,154.291
C04978=1079.000,220.068,421.146,174.819,25.064,154.292
C04979=1079.007,220.316,421.121,174.821,25.068,154.292
C04980=1079.012,220.566,421.096,174.823,25.071,154.293
C04981=1079.017,220.814,421.071,174.825,25.074,154.293
C04982=1079.024,221.063,421.045,174.828,25.078,154.294
C04983=1079.029,221.312,421.019,174.830,25.082,154.294
C04984=1079.035,221.560,420.994,174.832,25.085,154.295
C04985=1079.044,221.967,420.952,174.836,25.091,154.295
C04986=1079.054,222.374,420.910,174.839,25.096,154.296
C04987=1079.062,222.781,420.869,174.844,25.102,154.297
C04988=1079.072,223.187,420.827,174.847,25.108,154.298
C04989=1079.077,223.436,420.801,174.850,25.111,154.298
C04990=1079.083,223.685,420.776,174.852,25.115,154.299
C04991=1079.089,223.934,420.750,174.855,25.118,154.299
C04992=1079.095,224.182,420.724,174.857,25.122,154.299
C04993=1079.100,224.431,420.699,174.859,25.125,154.300
C04994=1079.106,224.679,420.673,174.861,25.129,154.300
C04995=1079.112,224.928,420.648,174.864,25.132,154.301
C04996=1079.118,225.176,420.621,174.866,25.136,154.301
C04997=1079.123,225.425,420.596,174.869,25.139,154.302
C04998=1079.129,225.674,420.570,174.871,25.143,154.302
C04999=1079.135,225.922,420.545,174.874,25.146,154.303
C05000=1079.140,226.171,420.519,174.876,25.150,154.303
C05001=1079.146,226.420,420.493,174.878,25.153,154.304
C05002=1079.152,226.668,420.467,174.880,25.157,154.304
C05003=1079.157,226.917,420.441,174.883,25.160,154.304
C05004=1079.163,227.165,420.416,174.885,25.164,154.305
C05005=1079.169,227.414,420.390,174.887,25.167,154.305
C05006=1079.175,227.663,420.365,174.890,25.171,154.306
C05007=1079.181,227.911,420.338,174.893,25.174,154.306
C05008=1079.186,228.160,420.312,174.895,25.177,154.307
C05009=1079.192,228.409,420.287,174.897,25.181,154.307
C05010=1079.198,228.657,420.260,174.899,25.184,154.308
C05011=1079.203,228.906,420.234,174.902,25.188,154.308
C05012=1079.209,229.154,420.209,174.904,25.191,154.308
C05013=1079.215,229.403,420.182,174.906,25.195,154.309
C05014=1079.220,229.652,420.156,174.909,25.198,154.309
C05015=1079.227,229.900,420.131,174.912,25.201,154.310
C05016=1079.232,230.149,420.104,174.914,25.205,154.310
C05017=1079.238,230.398,420.079,174.916,25.208,154.311
C05018=1079.244,230.646,420.053,174.918,25.212,154.311
C05019=1079.250,230.895,420.027,174.921,25.215,154.312
C05020=1079.255,231.144,420.001,174.923,25.219,154.312
C05021=1079.261,231.392,419.974,174.925,25.222,154.313
C05022=1079.266,231.640,419.948,174.928,25.226,154.313
C05023=1079.272,231.889,419.922,174.931,25.229,154.313
C05024=1079.278,232.137,419.896,174.933,25.233,154.314
C05025=1079.284,232.386,419.870,174.935,25.236,154.314
C05026=1079.289,232.635,419.844,174.938,25.240,154.315
C05027=1079.295,232.883,419.817,174.940,25.243,154.315
C05028=1079.300,233.132,419.791,174.942,25.247,154.316
C05029=1079.306,233.380,419.765,174.944,25.250,154.316
C05030=1079.312,233.629,419.739,174.947,25.254,154.317
C05031=1079.318,233.877,419.713,174.950,25.257,154.317
C05032=1079.324,234.126,419.687,174.952,25.261,154.318
C05033=1079.329,234.375,419.660,174.955,25.264,154.318
C05034=1079.335,234.624,419.634,174.957,25.268,154.319
C05035=1079.341,234.872,419.607,174.959,25.271,154.319
C05036=1079.346,235.120,419.581,174.962,25.275,154.319
C05037=1079.355,235.518,419.539,174.966,25.281,154.320
C05038=1079.364,235.917,419.496,174.969,25.286,154.321
C05039=1079.373,236.315,419.454,174.973,25.292,154.322
C05040=1079.383,236.714,419.412,174.978,25.298,154.322
C05041=1079.388,236.962,419.385,174.980,25.301,154.323
C05042=1079.394,237.211,419.359,174.982,25.304,154.323
C05043=1079.400,237.460,419.333,174.985,25.308,154.324
C05044=1079.405,237.708,419.306,174.987,25.312,154.324
C05045=1079.411,237.957,419.279,174.989,25.315,154.325
C05046=1079.417,238.205,419.253,174.992,25.319,154.325
C05047=1079.423,238.453,419.226,174.995,25.322,154.326
C05048=1079.428,238.702,419.200,174.997,25.325,154.326
C05049=1079.435,238.951,419.173,175.000,25.329,154.327
C05050=1079.440,239.200,419.146,175.002,25.333,154.327
C05051=1079.446,239.448,419.120,175.004,25.336,154.327
C05052=1079.452,239.696,419.093,175.007,25.340,154.328
C05053=1079.457,239.945,419.066,175.009,25.343,154.328
C05054=1079.463,240.193,419.039,175.011,25.346,154.329
C05055=1079.468,240.442,419.013,175.015,25.350,154.329
C05056=1079.474,240.691,418.987,175.017,25.354,154.330
C05057=1079.480,240.939,418.960,175.019,25.357,154.330
C05058=1079.486,241.188,418.933,175.022,25.361,154.331
C05059=1079.492,241.437,418.906,175.024,25.364,154.331
C05060=1079.498,241.685,418.880,175.026,25.367,154.332
C05061=1079.503,241.933,418.853,175.029,25.371,154.332
C05062=1079.508,242.182,418.826,175.031,25.375,154.333
C05063=1079.514,242.430,418.799,175.034,25.378,154.333
C05064=1079.520,242.679,418.772,175.037,25.381,154.333
C05065=1079.526,242.928,418.745,175.039,25.385,154.334
C05066=1079.532,243.176,418.719,175.041,25.388,154.334
C05067=1079.537,243.425,418.692,175.044,25.392,154.335
C05068=1079.543,243.673,418.665,175.046,25.396,154.335
C05069=1079.549,243.921,418.638,175.048,25.399,154.336
C05070=1079.555,244.169,418.611,175.051,25.403,154.336
C05071=1079.560,244.419,418.583,175.054,25.406,154.337
C05072=1079.566,244.667,418.557,175.056,25.409,154.337
C05073=1079.572,244.915,418.530,175.059,25.413,154.338
C05074=1079.577,245.164,418.503,175.061,25.416,154.338
C05075=1079.583,245.412,418.476,175.064,25.420,154.338
C05076=1079.589,245.660,418.449,175.066,25.424,154.339
C05077=1079.595,245.909,418.421,175.068,25.427,154.340
C05078=1079.600,246.158,418.394,175.072,25.431,154.340
C05079=1079.606,246.406,418.368,175.074,25.434,154.340
C05080=1079.611,246.655,418.341,175.076,25.437,154.341
C05081=1079.618,246.903,418.313,175.079,25.441,154.341
C05082=1079.623,247.152,418.286,175.081,25.445,154.342
C05083=1079.629,247.400,418.259,175.084,25.449,154.342
C05084=1079.634,247.648,418.231,175.086,25.452,154.343
C05085=1079.640,247.897,418.204,175.088,25.455,154.343
C05086=1079.645,248.146,418.177,175.092,25.459,154.344
C05087=1079.651,248.394,418.150,175.094,25.462,154.344
C05088=1079.656,248.642,418.122,175.096,25.466,154.345
C05089=1079.665,249.034,418.079,175.100,25.472,154.345
C05090=1079.675,249.426,418.037,175.104,25.478,154.346
C05091=1079.683,249.818,417.993,175.109,25.483,154.347
C05092=1079.692,250.209,417.950,175.112,25.489,154.348
C05093=1079.698,250.457,417.922,175.114,25.492,154.348
C05094=1079.703,250.706,417.895,175.117,25.496,154.349
C05095=1079.709,250.954,417.867,175.120,25.499,154.349
C05096=1079.715,251.203,417.840,175.122,25.503,154.350
C05097=1079.720,251.451,417.812,175.125,25.506,154.350
C05098=1079.726,251.700,417.786,175.127,25.510,154.350
C05099=1079.731,251.948,417.758,175.130,25.514,154.351
C05100=1079.737,252.197,417.730,175.132,25.517,154.351
C05101=1079.743,252.445,417.703,175.135,25.521,154.352
C05102=1079.748,252.693,417.675,175.138,25.524,154.352
C05103=1079.755,252.942,417.648,175.140,25.528,154.353
C05104=1079.760,253.190,417.620,175.143,25.532,154.353
C05105=1079.765,253.439,417.592,175.145,25.535,154.354
C05106=1079.772,253.687,417.565,175.148,25.539,154.354
C05107=1079.777,253.936,417.537,175.150,25.542,154.355
C05108=1079.783,254.184,417.509,175.152,25.546,154.355
C05109=1079.789,254.432,417.482,175.155,25.550,154.356
C05110=1079.794,254.681,417.455,175.158,25.553,154.356
C05111=1079.800,254.930,417.426,175.161,25.557,154.357
C05112=1079.806,255.177,417.399,175.163,25.560,154.357
C05113=1079.811,255.426,417.372,175.166,25.564,154.358
C05114=1079.817,255.675,417.343,175.168,25.567,154.358
C05115=1079.823,255.922,417.316,175.171,25.571,154.358
C05116=1079.829,256.171,417.288,175.173,25.574,154.359
C05117=1079.834,256.420,417.260,175.176,25.577,154.359
C05118=1079.841,256.668,417.233,175.179,25.581,154.360
C05119=1079.846,256.916,417.205,175.181,25.585,154.360
C05120=1079.851,257.164,417.177,175.184,25.589,154.361
C05121=1079.858,257.413,417.149,175.186,25.592,154.361
C05122=1079.863,257.662,417.122,175.189,25.596,154.362
C05123=1079.869,257.910,417.093,175.191,25.599,154.362
C05124=1079.874,258.158,417.065,175.195,25.603,154.363
C05125=1079.881,258.407,417.038,175.197,25.606,154.363
C05126=1079.887,258.655,417.010,175.199,25.609,154.364
C05127=1079.892,258.904,416.981,175.202,25.613,154.364
C05128=1079.899,259.151,416.954,175.204,25.616,154.365
C05129=1079.904,259.400,416.926,175.207,25.620,154.365
C05130=1079.910,259.648,416.898,175.209,25.623,154.365
C05131=1079.916,259.897,416.869,175.213,25.627,154.366
C05132=1079.922,260.145,416.842,175.215,25.630,154.366
C05133=1079.928,260.393,416.814,175.218,25.634,154.367
C05134=1079.934,260.642,416.785,175.220,25.638,154.367
C05135=1079.939,260.890,416.757,175.223,25.641,154.368
C05136=1079.946,261.139,416.730,175.225,25.645,154.368
C05137=1079.951,261.387,416.702,175.228,25.649,154.369
C05138=1079.957,261.635,416.673,175.231,25.652,154.369
C05139=1079.962,261.883,416.646,175.234,25.656,154.370
C05140=1079.968,262.132,416.617,175.236,25.659,154.370
C05141=1079.978,262.522,416.573,175.240,25.665,154.371
C05142=1079.987,262.910,416.529,175.244,25.670,154.372
C05143=1079.997,263.299,416.485,175.248,25.676,154.372
C05144=1080.006,263.688,416.442,175.253,25.681,154.373
C05145=1080.012,263.937,416.413,175.255,25.684,154.373
C05146=1080.017,264.184,416.385,175.258,25.688,154.374
C05147=1080.023,264.433,416.356,175.260,25.692,154.374
C05148=1080.029,264.682,416.328,175.263,25.695,154.375
C05149=1080.035,264.930,416.300,175.265,25.699,154.375
C05150=1080.041,265.178,416.271,175.268,25.703,154.376
C05151=1080.045,265.426,416.242,175.270,25.706,154.376
C05152=1080.051,265.675,416.214,175.274,25.710,154.377
C05153=1080.057,265.924,416.186,175.276,25.713,154.377
C05154=1080.063,266.171,416.157,175.279,25.717,154.378
C05155=1080.069,266.420,416.129,175.281,25.720,154.378
C05156=1080.074,266.668,416.101,175.284,25.724,154.379
C05157=1080.080,266.916,416.072,175.287,25.728,154.379
C05158=1080.086,267.165,416.043,175.290,25.731,154.380
C05159=1080.092,267.412,416.015,175.293,25.735,154.380
C05160=1080.098,267.661,415.986,175.295,25.739,154.381
C05161=1080.103,267.910,415.957,175.298,25.742,154.381
C05162=1080.109,268.157,415.929,175.300,25.746,154.382
C05163=1080.115,268.406,415.900,175.303,25.750,154.382
C05164=1080.121,268.654,415.871,175.305,25.753,154.383
C05165=1080.126,268.902,415.843,175.308,25.757,154.383
C05166=1080.133,269.150,415.814,175.311,25.761,154.384
C05167=1080.139,269.399,415.786,175.314,25.764,154.384
C05168=1080.143,269.647,415.757,175.316,25.768,154.385
C05169=1080.149,269.896,415.729,175.319,25.771,154.385
C05170=1080.156,270.144,415.699,175.321,25.775,154.386
C05171=1080.162,270.393,415.671,175.324,25.778,154.386
C05172=1080.167,270.640,415.642,175.326,25.782,154.387
C05173=1080.173,270.888,415.613,175.329,25.786,154.387
C05174=1080.179,271.137,415.585,175.333,25.790,154.388
C05175=1080.184,271.385,415.556,175.335,25.793,154.388
C05176=1080.190,271.634,415.527,175.338,25.797,154.388
C05177=1080.196,271.882,415.498,175.340,25.801,154.389
C05178=1080.202,272.130,415.469,175.343,25.804,154.390
C05179=1080.207,272.378,415.440,175.345,25.808,154.390
C05180=1080.213,272.626,415.411,175.348,25.811,154.390
C05181=1080.219,272.875,415.382,175.351,25.815,154.391
C05182=1080.224,273.124,415.353,175.354,25.819,154.391
C05183=1080.230,273.371,415.325,175.357,25.822,154.392
C05184=1080.236,273.619,415.296,175.359,25.826,154.392
C05185=1080.242,273.868,415.266,175.362,25.830,154.393
C05186=1080.248,274.116,415.238,175.364,25.834,154.393
C05187=1080.254,274.364,415.209,175.367,25.837,154.394
C05188=1080.259,274.612,415.179,175.370,25.841,154.394
C05189=1080.265,274.860,415.150,175.373,25.844,154.395
C05190=1080.271,275.109,415.121,175.375,25.848,154.395
C05191=1080.277,275.357,415.092,175.378,25.852,154.396
C05192=1080.282,275.606,415.063,175.381,25.856,154.396
C05193=1080.292,276.020,415.014,175.385,25.862,154.397
C05194=1080.301,276.435,414.966,175.390,25.868,154.398
C05195=1080.311,276.850,414.917,175.395,25.874,154.399
C05196=1080.321,277.264,414.868,175.399,25.880,154.400
C05197=1080.326,277.513,414.838,175.401,25.884,154.400
C05198=1080.333,277.761,414.809,175.405,25.887,154.401
C05199=1080.338,278.009,414.779,175.407,25.891,154.401
C05200=1080.344,278.257,414.750,175.410,25.895,154.402
C05201=1080.349,278.505,414.721,175.413,25.899,154.402
C05202=1080.356,278.753,414.692,175.415,25.902,154.403
C05203=1080.361,279.002,414.662,175.418,25.906,154.403
C05204=1080.367,279.250,414.633,175.420,25.910,154.404
C05205=1080.373,279.498,414.604,175.423,25.913,154.404
C05206=1080.378,279.747,414.574,175.427,25.917,154.405
C05207=1080.385,279.995,414.545,175.429,25.921,154.405
C05208=1080.390,280.243,414.515,175.432,25.925,154.406
C05209=1080.396,280.491,414.486,175.434,25.928,154.406
C05210=1080.402,280.739,414.456,175.437,25.932,154.407
C05211=1080.408,280.987,414.427,175.440,25.936,154.407
C05212=1080.413,281.235,414.398,175.442,25.939,154.408
C05213=1080.419,281.484,414.368,175.445,25.943,154.408
C05214=1080.424,281.732,414.338,175.448,25.947,154.409
C05215=1080.431,281.979,414.309,175.451,25.951,154.409
C05216=1080.436,282.228,414.279,175.454,25.954,154.410
C05217=1080.442,282.476,414.249,175.456,25.958,154.410
C05218=1080.447,282.725,414.220,175.459,25.962,154.411
C05219=1080.454,282.972,414.190,175.462,25.966,154.411
C05220=1080.459,283.221,414.160,175.464,25.969,154.412
C05221=1080.465,283.469,414.131,175.467,25.973,154.412
C05222=1080.471,283.717,414.100,175.470,25.977,154.413
C05223=1080.476,283.965,414.071,175.473,25.981,154.414
C05224=1080.483,284.214,414.042,175.476,25.985,154.414
C05225=1080.488,284.461,414.011,175.478,25.988,154.415
C05226=1080.494,284.710,413.982,175.481,25.992,154.415
C05227=1080.500,284.958,413.951,175.484,25.996,154.416
C05228=1080.505,285.206,413.922,175.486,26.000,154.416
C05229=1080.512,285.454,413.892,175.489,26.004,154.417
C05230=1080.517,285.702,413.862,175.492,26.007,154.417
C05231=1080.523,285.951,413.833,175.495,26.011,154.418
C05232=1080.529,286.198,413.802,175.498,26.015,154.418
C05233=1080.535,286.434,413.774,175.500,26.018,154.419
C05234=1080.539,286.671,413.746,175.503,26.022,154.419
C05235=1080.545,286.909,413.716,175.505,26.025,154.420
C05236=1080.551,287.145,413.689,175.508,26.029,154.420
C05237=1080.556,287.382,413.660,175.511,26.033,154.421
C05238=1080.561,287.618,413.631,175.514,26.036,154.421
C05239=1080.568,287.855,413.603,175.516,26.040,154.422
C05240=1080.573,288.092,413.574,175.519,26.044,154.422
C05241=1080.579,288.340,413.543,175.522,26.048,154.423
C05242=1080.584,288.588,413.514,175.524,26.051,154.423
C05243=1080.591,288.836,413.484,175.527,26.055,154.424
C05244=1080.597,289.084,413.453,175.530,26.059,154.424
C05245=1080.606,289.486,413.405,175.535,26.065,154.425
C05246=1080.615,289.887,413.356,175.540,26.071,154.426
C05247=1080.625,290.289,413.307,175.544,26.077,154.427
C05248=1080.635,290.691,413.258,175.549,26.084,154.428
C05249=1080.640,290.940,413.228,175.551,26.087,154.428
C05250=1080.646,291.187,413.198,175.554,26.091,154.429
C05251=1080.652,291.435,413.167,175.557,26.095,154.429
C05252=1080.657,291.683,413.136,175.559,26.099,154.430
C05253=1080.663,291.931,413.106,175.562,26.103,154.430
C05254=1080.668,292.180,413.076,175.566,26.107,154.431
C05255=1080.675,292.428,413.046,175.568,26.111,154.432
C05256=1080.681,292.676,413.015,175.571,26.115,154.432
C05257=1080.686,292.924,412.985,175.574,26.118,154.433
C05258=1080.692,293.172,412.955,175.577,26.122,154.433
C05259=1080.698,293.419,412.924,175.579,26.126,154.434
C05260=1080.704,293.667,412.894,175.582,26.130,154.434
C05261=1080.709,293.916,412.863,175.585,26.134,154.435
C05262=1080.715,294.164,412.832,175.587,26.138,154.435
C05263=1080.721,294.412,412.802,175.590,26.142,154.436
C05264=1080.727,294.660,412.772,175.594,26.145,154.436
C05265=1080.733,294.907,412.741,175.597,26.149,154.437
C05266=1080.739,295.156,412.711,175.599,26.153,154.438
C05267=1080.744,295.404,412.680,175.602,26.157,154.438
C05268=1080.750,295.652,412.649,175.605,26.161,154.439
C05269=1080.756,295.900,412.619,175.608,26.165,154.439
C05270=1080.762,296.148,412.588,175.610,26.169,154.440
C05271=1080.768,296.396,412.558,175.613,26.172,154.440
C05272=1080.773,296.644,412.527,175.616,26.177,154.441
C05273=1080.779,296.892,412.497,175.620,26.181,154.441
C05274=1080.786,297.140,412.465,175.622,26.184,154.442
C05275=1080.791,297.388,412.434,175.625,26.188,154.442
C05276=1080.797,297.636,412.404,175.628,26.192,154.443
C05277=1080.803,297.884,412.373,175.631,26.196,154.444
C05278=1080.808,298.133,412.342,175.633,26.200,154.444
C05279=1080.814,298.380,412.311,175.636,26.204,154.445
C05280=1080.819,298.628,412.280,175.639,26.208,154.445
C05281=1080.825,298.876,412.250,175.642,26.213,154.446
C05282=1080.831,299.125,412.219,175.644,26.216,154.447
C05283=1080.837,299.372,412.187,175.648,26.220,154.447
C05284=1080.842,299.620,412.157,175.651,26.224,154.448
C05285=1080.848,299.868,412.126,175.654,26.228,154.448
C05286=1080.854,300.116,412.094,175.656,26.232,154.449
C05287=1080.860,300.364,412.064,175.659,26.236,154.449
C05288=1080.865,300.612,412.033,175.662,26.241,154.450
C05289=1080.871,300.860,412.001,175.665,26.244,154.451
C05290=1080.877,301.108,411.970,175.667,26.248,154.451
C05291=1080.883,301.355,411.939,175.670,26.252,154.452
C05292=1080.888,301.603,411.908,175.673,26.256,154.452
C05293=1080.894,301.852,411.878,175.676,26.261,154.453
C05294=1080.900,302.099,411.846,175.680,26.264,154.453
C05295=1080.905,302.347,411.815,175.682,26.268,154.454
C05296=1080.911,302.595,411.784,175.685,26.272,154.455
C05297=1080.920,303.012,411.731,175.690,26.280,154.456
C05298=1080.930,303.427,411.679,175.695,26.286,154.457
C05299=1080.940,303.843,411.627,175.699,26.293,154.458
C05300=1080.949,304.259,411.574,175.705,26.300,154.459
C05301=1080.956,304.507,411.543,175.708,26.304,154.459
C05302=1080.961,304.755,411.511,175.710,26.308,154.460
C05303=1080.967,305.004,411.480,175.713,26.312,154.460
C05304=1080.973,305.251,411.449,175.716,26.316,154.461
C05305=1080.978,305.499,411.417,175.719,26.320,154.462
C05306=1080.985,305.746,411.386,175.722,26.324,154.462
C05307=1080.990,305.995,411.355,175.725,26.328,154.463
C05308=1080.996,306.243,411.323,175.727,26.332,154.463
C05309=1081.002,306.490,411.292,175.730,26.336,154.464
C05310=1081.008,306.739,411.261,175.733,26.340,154.465
C05311=1081.013,306.986,411.229,175.736,26.344,154.465
C05312=1081.020,307.234,411.197,175.740,26.348,154.466
C05313=1081.026,307.482,411.166,175.743,26.353,154.466
C05314=1081.032,307.730,411.134,175.745,26.357,154.467
C05315=1081.037,307.978,411.103,175.748,26.361,154.468
C05316=1081.043,308.226,411.071,175.751,26.365,154.468
C05317=1081.049,308.474,411.040,175.754,26.369,154.469
C05318=1081.055,308.721,411.008,175.757,26.373,154.469
C05319=1081.061,308.969,410.977,175.760,26.377,154.470
C05320=1081.067,309.217,410.945,175.762,26.381,154.471
C05321=1081.073,309.465,410.913,175.765,26.385,154.471
C05322=1081.079,309.713,410.881,175.768,26.389,154.472
C05323=1081.085,309.961,410.850,175.772,26.394,154.472
C05324=1081.090,310.209,410.819,175.775,26.397,154.473
C05325=1081.096,310.457,410.786,175.778,26.402,154.474
C05326=1081.103,310.705,410.755,175.781,26.406,154.474
C05327=1081.108,310.953,410.723,175.784,26.410,154.475
C05328=1081.114,311.201,410.691,175.786,26.414,154.475
C05329=1081.120,311.449,410.659,175.789,26.418,154.476
C05330=1081.126,311.696,410.628,175.792,26.422,154.477
C05331=1081.133,311.944,410.596,175.795,26.426,154.477
C05332=1081.139,312.192,410.564,175.798,26.430,154.478
C05333=1081.144,312.439,410.532,175.801,26.435,154.478
C05334=1081.151,312.687,410.500,175.805,26.439,154.479
C05335=1081.157,312.936,410.468,175.808,26.443,154.480
C05336=1081.162,313.183,410.437,175.810,26.447,154.480
C05337=1081.168,313.431,410.405,175.813,26.451,154.481
C05338=1081.174,313.680,410.373,175.816,26.455,154.481
C05339=1081.181,313.927,410.341,175.819,26.459,154.482
C05340=1081.186,314.174,410.309,175.822,26.463,154.483
C05341=1081.192,314.423,410.277,175.825,26.468,154.483
C05342=1081.198,314.671,410.245,175.828,26.472,154.484
C05343=1081.204,314.919,410.213,175.831,26.476,154.484
C05344=1081.210,315.166,410.180,175.834,26.480,154.485
C05345=1081.216,315.414,410.148,175.836,26.484,154.486
C05346=1081.221,315.663,410.116,175.839,26.489,154.486
C05347=1081.227,315.909,410.083,175.843,26.493,154.487
C05348=1081.233,316.158,410.051,175.846,26.497,154.488
C05349=1081.242,316.577,409.997,175.851,26.505,154.489
C05350=1081.252,316.996,409.942,175.855,26.512,154.490
C05351=1081.262,317.415,409.888,175.861,26.519,154.491
C05352=1081.272,317.834,409.832,175.866,26.527,154.492
C05353=1081.277,318.082,409.800,175.869,26.531,154.493
C05354=1081.283,318.330,409.768,175.871,26.535,154.493
C05355=1081.289,318.578,409.735,175.874,26.539,154.494
C05356=1081.294,318.825,409.703,175.877,26.544,154.495
C05357=1081.301,319.073,409.671,175.880,26.549,154.496
C05358=1081.307,319.321,409.639,175.883,26.553,154.496
C05359=1081.312,319.569,409.605,175.886,26.557,154.497
C05360=1081.318,319.817,409.572,175.889,26.562,154.497
C05361=1081.324,320.064,409.541,175.892,26.566,154.498
C05362=1081.329,320.312,409.507,175.896,26.570,154.499
C05363=1081.335,320.560,409.475,175.899,26.575,154.499
C05364=1081.342,320.808,409.443,175.902,26.579,154.500
C05365=1081.347,321.056,409.409,175.905,26.584,154.501
C05366=1081.353,321.304,409.377,175.908,26.588,154.502
C05367=1081.359,321.551,409.345,175.911,26.592,154.502
C05368=1081.364,321.799,409.312,175.914,26.597,154.503
C05369=1081.370,322.047,409.280,175.917,26.601,154.503
C05370=1081.377,322.295,409.247,175.920,26.605,154.504
C05371=1081.382,322.542,409.213,175.922,26.610,154.505
C05372=1081.388,322.790,409.181,175.925,26.614,154.506
C05373=1081.394,323.038,409.149,175.928,26.618,154.506
C05374=1081.400,323.286,409.115,175.931,26.623,154.507
C05375=1081.406,323.534,409.083,175.934,26.627,154.508
C05376=1081.412,323.781,409.050,175.937,26.632,154.508
C05377=1081.418,324.029,409.017,175.940,26.636,154.509
C05378=1081.424,324.277,408.985,175.943,26.641,154.510
C05379=1081.429,324.525,408.952,175.946,26.645,154.510
C05380=1081.435,324.772,408.919,175.949,26.649,154.511
C05381=1081.442,325.020,408.886,175.952,26.654,154.512
C05382=1081.447,325.268,408.853,175.955,26.658,154.512
C05383=1081.454,325.515,408.820,175.958,26.663,154.513
C05384=1081.459,325.763,408.787,175.962,26.667,154.514
C05385=1081.465,326.011,408.754,175.965,26.672,154.514
C05386=1081.471,326.259,408.721,175.968,26.676,154.515
C05387=1081.477,326.506,408.688,175.971,26.680,154.516
C05388=1081.483,326.754,408.654,175.974,26.685,154.517
C05389=1081.489,327.002,408.622,175.977,26.689,154.517
C05390=1081.495,327.249,408.589,175.980,26.694,154.518
C05391=1081.501,327.497,408.556,175.983,26.699,154.519
C05392=1081.508,327.746,408.523,175.986,26.703,154.519
C05393=1081.513,327.994,408.489,175.989,26.707,154.520
C05394=1081.520,328.241,408.456,175.992,26.712,154.521
C05395=1081.525,328.489,408.423,175.995,26.716,154.521
C05396=1081.532,328.736,408.390,175.999,26.721,154.522
C05397=1081.537,328.984,408.356,176.002,26.726,154.523
C05398=1081.544,329.231,408.324,176.005,26.730,154.523
C05399=1081.549,329.479,408.290,176.008,26.734,154.524
C05400=1081.556,329.727,408.258,176.011,26.739,154.525
C05401=1081.565,330.140,408.202,176.016,26.746,154.526
C05402=1081.575,330.552,408.146,176.021,26.754,154.527
C05403=1081.585,330.965,408.091,176.026,26.762,154.528
C05404=1081.596,331.377,408.036,176.032,26.769,154.530
C05405=1081.603,331.625,408.001,176.035,26.774,154.530
C05406=1081.608,331.873,407.968,176.038,26.778,154.531
C05407=1081.614,332.120,407.935,176.041,26.783,154.532
C05408=1081.620,332.368,407.901,176.044,26.788,154.533
C05409=1081.626,332.616,407.868,176.047,26.792,154.533
C05410=1081.631,332.863,407.834,176.050,26.797,154.534
C05411=1081.637,333.111,407.800,176.053,26.801,154.535
C05412=1081.643,333.359,407.767,176.056,26.806,154.536
C05413=1081.650,333.606,407.733,176.059,26.811,154.536
C05414=1081.656,333.854,407.700,176.063,26.816,154.537
C05415=1081.661,334.101,407.666,176.066,26.820,154.538
C05416=1081.667,334.349,407.632,176.069,26.825,154.538
C05417=1081.673,334.597,407.598,176.072,26.830,154.539
C05418=1081.679,334.845,407.564,176.075,26.835,154.540
C05419=1081.685,335.093,407.531,176.078,26.840,154.541
C05420=1081.691,335.340,407.497,176.081,26.844,154.541
C05421=1081.697,335.587,407.464,176.084,26.849,154.542
C05422=1081.703,335.835,407.429,176.087,26.853,154.543
C05423=1081.709,336.083,407.395,176.090,26.858,154.544
C05424=1081.715,336.331,407.362,176.094,26.863,154.545
C05425=1081.721,336.578,407.328,176.097,26.868,154.545
C05426=1081.727,336.826,407.293,176.100,26.872,154.546
C05427=1081.733,337.074,407.260,176.103,26.877,154.547
C05428=1081.739,337.321,407.226,176.106,26.882,154.548
C05429=1081.745,337.569,407.192,176.109,26.887,154.548
C05430=1081.751,337.816,407.158,176.112,26.892,154.549
C05431=1081.757,338.064,407.125,176.116,26.897,154.550
C05432=1081.762,338.312,407.090,176.119,26.901,154.551
C05433=1081.769,338.560,407.056,176.122,26.906,154.552
C05434=1081.775,338.807,407.022,176.125,26.911,154.552
C05435=1081.781,339.054,406.988,176.128,26.916,154.553
C05436=1081.787,339.302,406.953,176.131,26.921,154.554
C05437=1081.793,339.550,406.920,176.134,26.926,154.555
C05438=1081.798,339.797,406.886,176.137,26.931,154.556
C05439=1081.805,340.045,406.851,176.140,26.936,154.556
C05440=1081.811,340.293,406.817,176.143,26.940,154.557
C05441=1081.816,340.540,406.783,176.146,26.945,154.558
C05442=1081.822,340.788,406.748,176.149,26.950,154.559
C05443=1081.828,341.035,406.714,176.152,26.955,154.560
C05444=1081.834,341.283,406.680,176.156,26.960,154.560
C05445=1081.840,341.531,406.646,176.159,26.965,154.561
C05446=1081.846,341.778,406.612,176.162,26.970,154.562
C05447=1081.853,342.026,406.577,176.165,26.975,154.563
C05448=1081.858,342.274,406.543,176.168,26.980,154.564
C05449=1081.864,342.520,406.508,176.172,26.985,154.564
C05450=1081.871,342.768,406.474,176.175,26.990,154.565
C05451=1081.876,343.015,406.439,176.178,26.994,154.566
C05452=1081.883,343.263,406.405,176.181,27.000,154.567
C05453=1081.892,343.670,406.349,176.186,27.008,154.568
C05454=1081.902,344.077,406.292,176.192,27.016,154.570
C05455=1081.912,344.484,406.235,176.197,27.024,154.571
C05456=1081.922,344.891,406.178,176.202,27.033,154.572
C05457=1081.928,345.139,406.144,176.205,27.038,154.573
